// Mitsubishi GX Works2 project: LG 250T Press 3 21.07.21   PLC: Q03UD
// LG 250T Press 3 21.07.21

PROGRAM MAIN
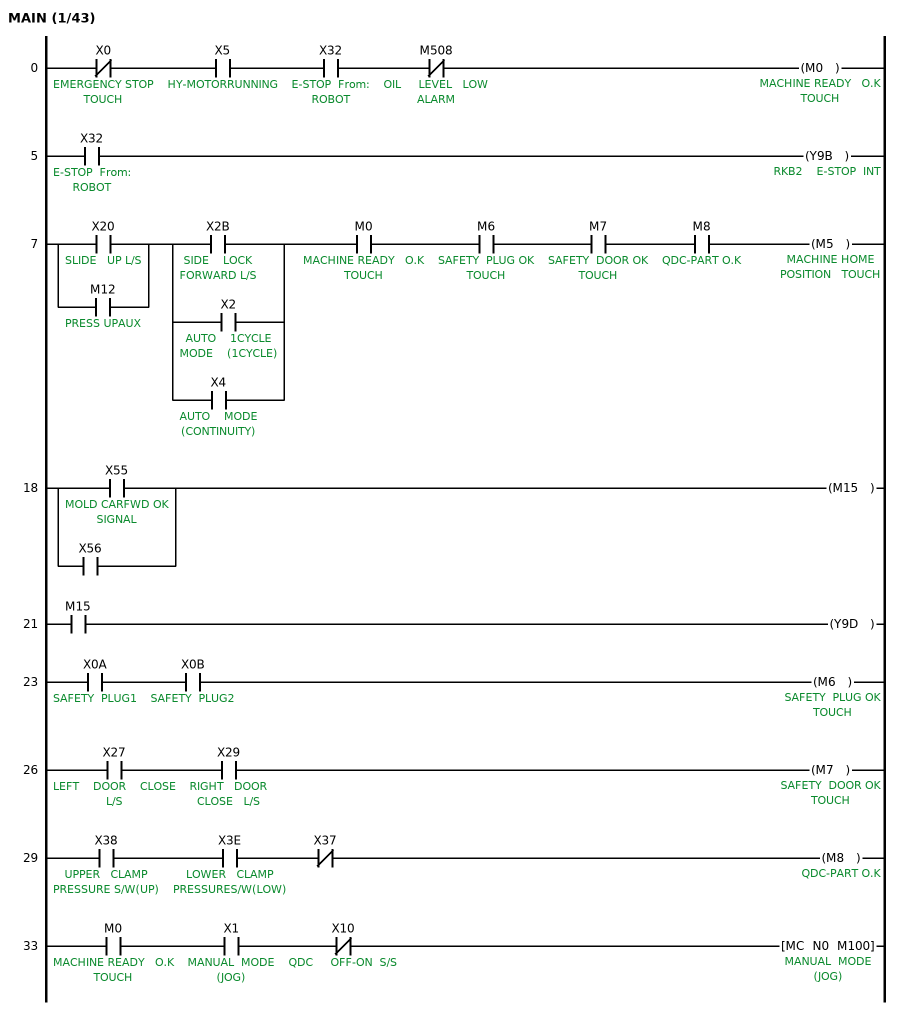
0     LDI     X0  ; EMERGENCY STOP  TOUCH
      AND     X5  ; HY-MOTORRUNNING
      AND     X32  ; E-STOP  From:   ROBOT
      ANI     M508  ; OIL     LEVEL   LOW     ALARM
      OUT     M0  ; MACHINE READY   O.K     TOUCH
5     LD      X32  ; E-STOP  From:   ROBOT
      OUT     Y9B  ; RKB2    E-STOP  INT
7     LD      X20  ; SLIDE   UP L/S
      OR      M12  ; PRESS UPAUX
      LD      X2B  ; SIDE    LOCK    FORWARD L/S
      OR      X2  ; AUTO    1CYCLE  MODE    (1CYCLE)
      OR      X4  ; AUTO    MODE    (CONTINUITY)
      ANB
      AND     M0  ; MACHINE READY   O.K     TOUCH
      AND     M6  ; SAFETY  PLUG OK TOUCH
      AND     M7  ; SAFETY  DOOR OK TOUCH
      AND     M8  ; QDC-PART O.K
      OUT     M5  ; MACHINE HOME POSITION   TOUCH
18    LD      X55  ; MOLD CARFWD OK  SIGNAL
      OR      X56
      OUT     M15
21    LD      M15
      OUT     Y9D
23    LD      X0A  ; SAFETY  PLUG1
      AND     X0B  ; SAFETY  PLUG2
      OUT     M6  ; SAFETY  PLUG OK TOUCH
26    LD      X27  ; LEFT    DOOR    CLOSE   L/S
      AND     X29  ; RIGHT   DOOR    CLOSE   L/S
      OUT     M7  ; SAFETY  DOOR OK TOUCH
29    LD      X38  ; UPPER   CLAMP   PRESSURE S/W(UP)
      AND     X3E  ; LOWER   CLAMP   PRESSURES/W(LOW)
      ANI     X37
      OUT     M8  ; QDC-PART O.K
33    LD      M0  ; MACHINE READY   O.K     TOUCH
      AND     X1  ; MANUAL  MODE    (JOG)
      ANI     X10  ; QDC     OFF-ON  S/S
      MC      N0 M100  ; MANUAL  MODE    (JOG)
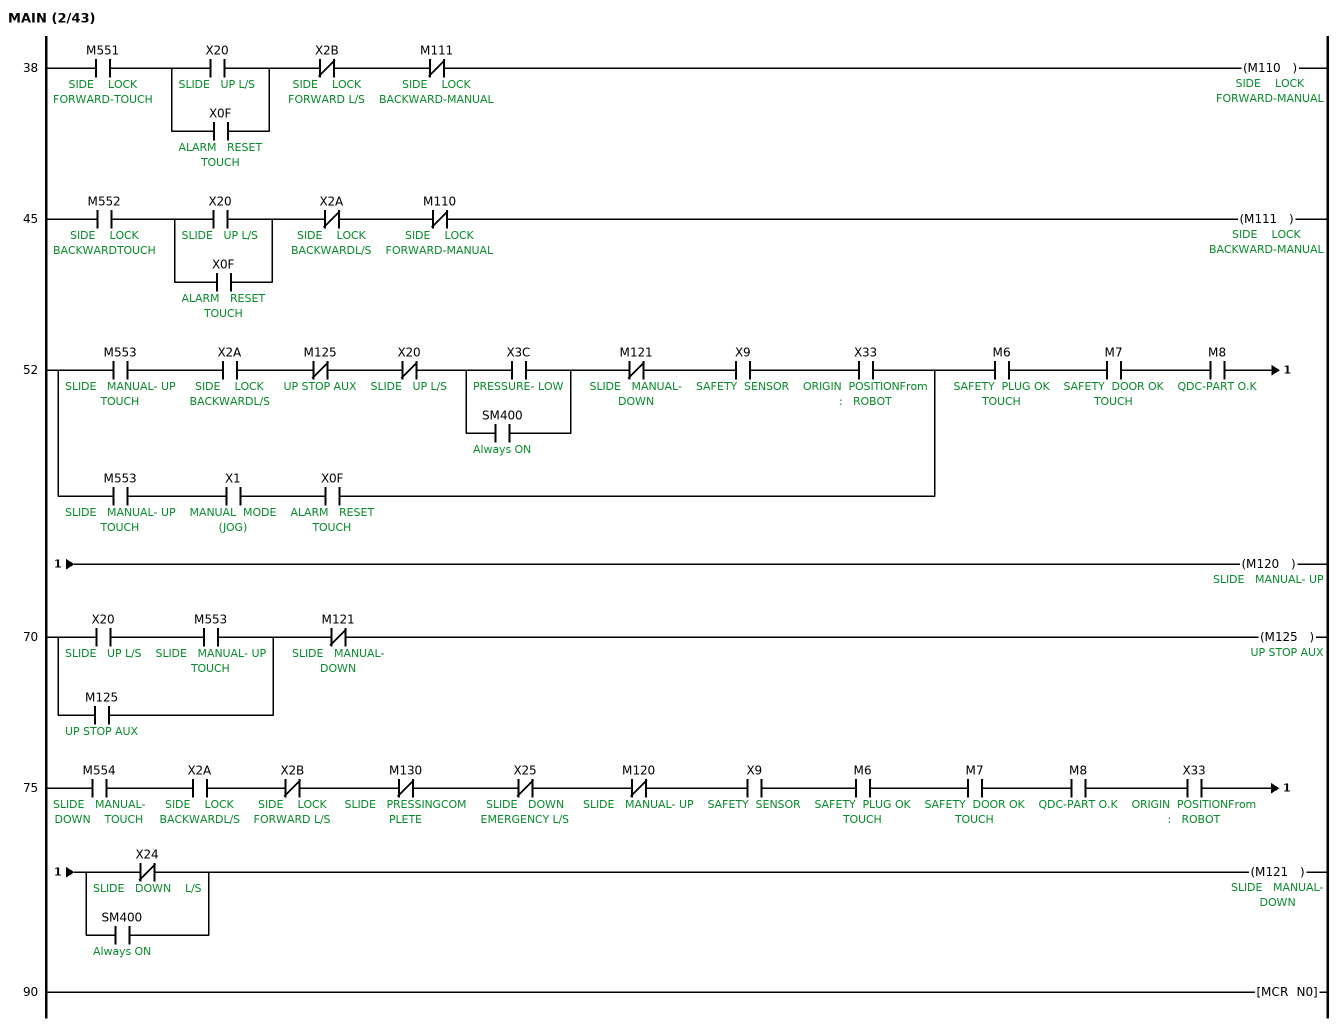
38    LD      M551  ; SIDE    LOCK    FORWARD-TOUCH
      LD      X20  ; SLIDE   UP L/S
      OR      X0F  ; ALARM   RESET   TOUCH
      ANB
      ANI     X2B  ; SIDE    LOCK    FORWARD L/S
      ANI     M111  ; SIDE    LOCK    BACKWARD-MANUAL
      OUT     M110  ; SIDE    LOCK    FORWARD-MANUAL
45    LD      M552  ; SIDE    LOCK    BACKWARDTOUCH
      LD      X20  ; SLIDE   UP L/S
      OR      X0F  ; ALARM   RESET   TOUCH
      ANB
      ANI     X2A  ; SIDE    LOCK    BACKWARDL/S
      ANI     M110  ; SIDE    LOCK    FORWARD-MANUAL
      OUT     M111  ; SIDE    LOCK    BACKWARD-MANUAL
52    LD      M553  ; SLIDE   MANUAL- UP      TOUCH
      AND     X2A  ; SIDE    LOCK    BACKWARDL/S
      ANI     M125  ; UP STOP AUX
      ANI     X20  ; SLIDE   UP L/S
      LD      X3C  ; PRESSURE- LOW
      OR      SM400  ; Always ON
      ANB
      ANI     M121  ; SLIDE   MANUAL- DOWN
      AND     X9  ; SAFETY  SENSOR
      AND     X33  ; ORIGIN  POSITIONFrom:   ROBOT
      LD      M553  ; SLIDE   MANUAL- UP      TOUCH
      AND     X1  ; MANUAL  MODE    (JOG)
      AND     X0F  ; ALARM   RESET   TOUCH
      ORB
      AND     M6  ; SAFETY  PLUG OK TOUCH
      AND     M7  ; SAFETY  DOOR OK TOUCH
      AND     M8  ; QDC-PART O.K
      OUT     M120  ; SLIDE   MANUAL- UP
70    LD      X20  ; SLIDE   UP L/S
      AND     M553  ; SLIDE   MANUAL- UP      TOUCH
      OR      M125  ; UP STOP AUX
      ANI     M121  ; SLIDE   MANUAL- DOWN
      OUT     M125  ; UP STOP AUX
75    LD      M554  ; SLIDE   MANUAL- DOWN    TOUCH
      AND     X2A  ; SIDE    LOCK    BACKWARDL/S
      ANI     X2B  ; SIDE    LOCK    FORWARD L/S
      ANI     M130  ; SLIDE   PRESSINGCOMPLETE
      ANI     X25  ; SLIDE   DOWN    EMERGENCY L/S
      ANI     M120  ; SLIDE   MANUAL- UP
      AND     X9  ; SAFETY  SENSOR
      AND     M6  ; SAFETY  PLUG OK TOUCH
      AND     M7  ; SAFETY  DOOR OK TOUCH
      AND     M8  ; QDC-PART O.K
      AND     X33  ; ORIGIN  POSITIONFrom:   ROBOT
      LDI     X24  ; SLIDE   DOWN    L/S
      OR      SM400  ; Always ON
      ANB
      OUT     M121  ; SLIDE   MANUAL- DOWN
90    MCR     N0
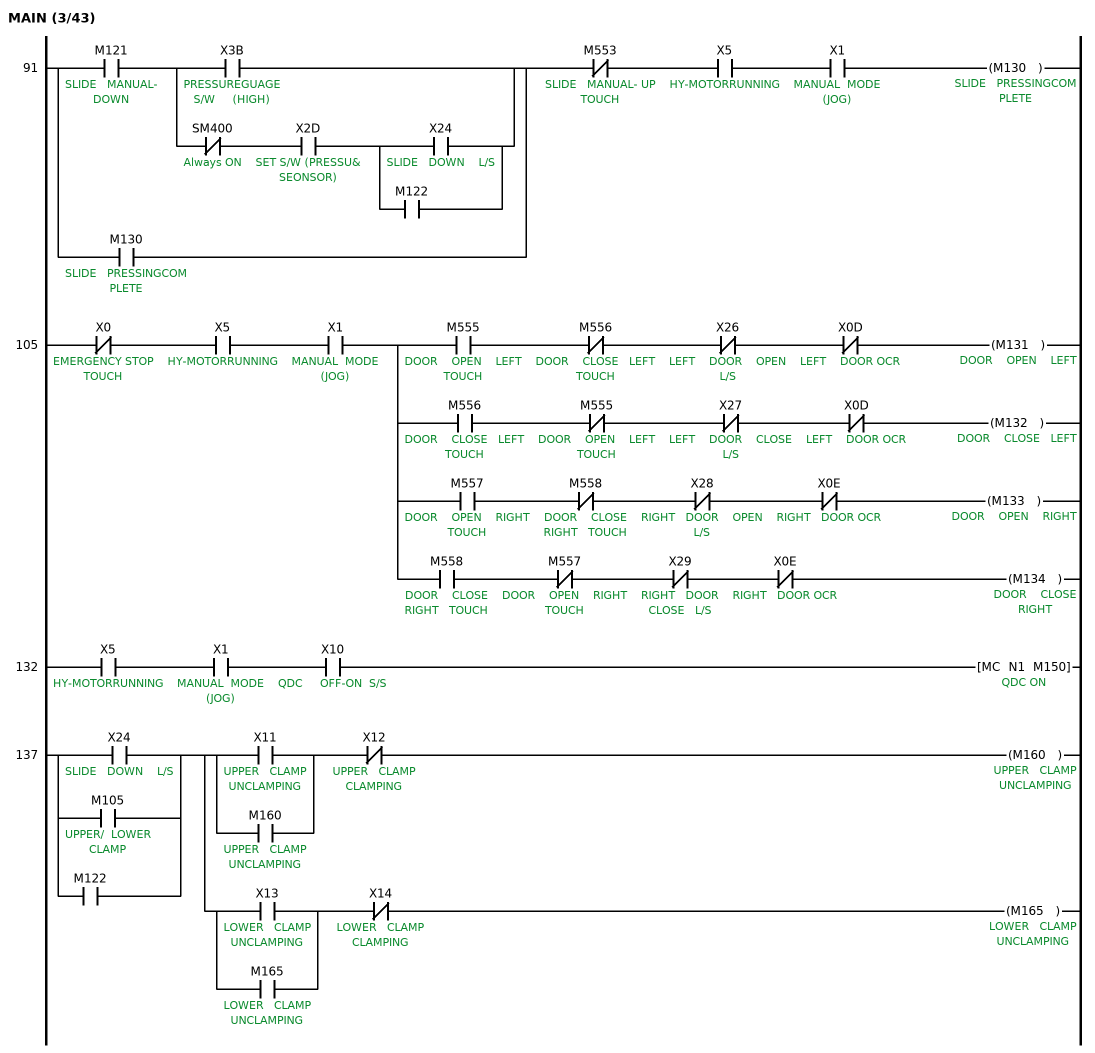
91    LD      M121  ; SLIDE   MANUAL- DOWN
      LD      X3B  ; PRESSUREGUAGE   S/W     (HIGH)
      LDI     SM400  ; Always ON
      AND     X2D  ; SET S/W (PRESSU& SEONSOR)
      LD      X24  ; SLIDE   DOWN    L/S
      OR      M122
      ANB
      ORB
      ANB
      OR      M130  ; SLIDE   PRESSINGCOMPLETE
      ANI     M553  ; SLIDE   MANUAL- UP      TOUCH
      AND     X5  ; HY-MOTORRUNNING
      AND     X1  ; MANUAL  MODE    (JOG)
      OUT     M130  ; SLIDE   PRESSINGCOMPLETE
105   LDI     X0  ; EMERGENCY STOP  TOUCH
      AND     X5  ; HY-MOTORRUNNING
      AND     X1  ; MANUAL  MODE    (JOG)
      MPS
      AND     M555  ; DOOR    OPEN    LEFT    TOUCH
      ANI     M556  ; DOOR    CLOSE   LEFT    TOUCH
      ANI     X26  ; LEFT    DOOR    OPEN L/S
      ANI     X0D  ; LEFT    DOOR OCR
      OUT     M131  ; DOOR    OPEN    LEFT
      MRD
      AND     M556  ; DOOR    CLOSE   LEFT    TOUCH
      ANI     M555  ; DOOR    OPEN    LEFT    TOUCH
      ANI     X27  ; LEFT    DOOR    CLOSE   L/S
      ANI     X0D  ; LEFT    DOOR OCR
      OUT     M132  ; DOOR    CLOSE   LEFT
      MRD
      AND     M557  ; DOOR    OPEN    RIGHT   TOUCH
      ANI     M558  ; DOOR    CLOSE   RIGHT   TOUCH
      ANI     X28  ; RIGHT   DOOR    OPEN L/S
      ANI     X0E  ; RIGHT   DOOR OCR
      OUT     M133  ; DOOR    OPEN    RIGHT
      MPP
      AND     M558  ; DOOR    CLOSE   RIGHT   TOUCH
      ANI     M557  ; DOOR    OPEN    RIGHT   TOUCH
      ANI     X29  ; RIGHT   DOOR    CLOSE   L/S
      ANI     X0E  ; RIGHT   DOOR OCR
      OUT     M134  ; DOOR    CLOSE   RIGHT
132   LD      X5  ; HY-MOTORRUNNING
      AND     X1  ; MANUAL  MODE    (JOG)
      AND     X10  ; QDC     OFF-ON  S/S
      MC      N1 M150  ; QDC ON
137   LD      X24  ; SLIDE   DOWN    L/S
      OR      M105  ; UPPER/  LOWER   CLAMP
      OR      M122
      MPS
      LD      X11  ; UPPER   CLAMP   UNCLAMPING
      OR      M160  ; UPPER   CLAMP   UNCLAMPING
      ANB
      ANI     X12  ; UPPER   CLAMP   CLAMPING
      OUT     M160  ; UPPER   CLAMP   UNCLAMPING
      MPP
      LD      X13  ; LOWER   CLAMP   UNCLAMPING
      OR      M165  ; LOWER   CLAMP   UNCLAMPING
      ANB
      ANI     X14  ; LOWER   CLAMP   CLAMPING
      OUT     M165  ; LOWER   CLAMP   UNCLAMPING
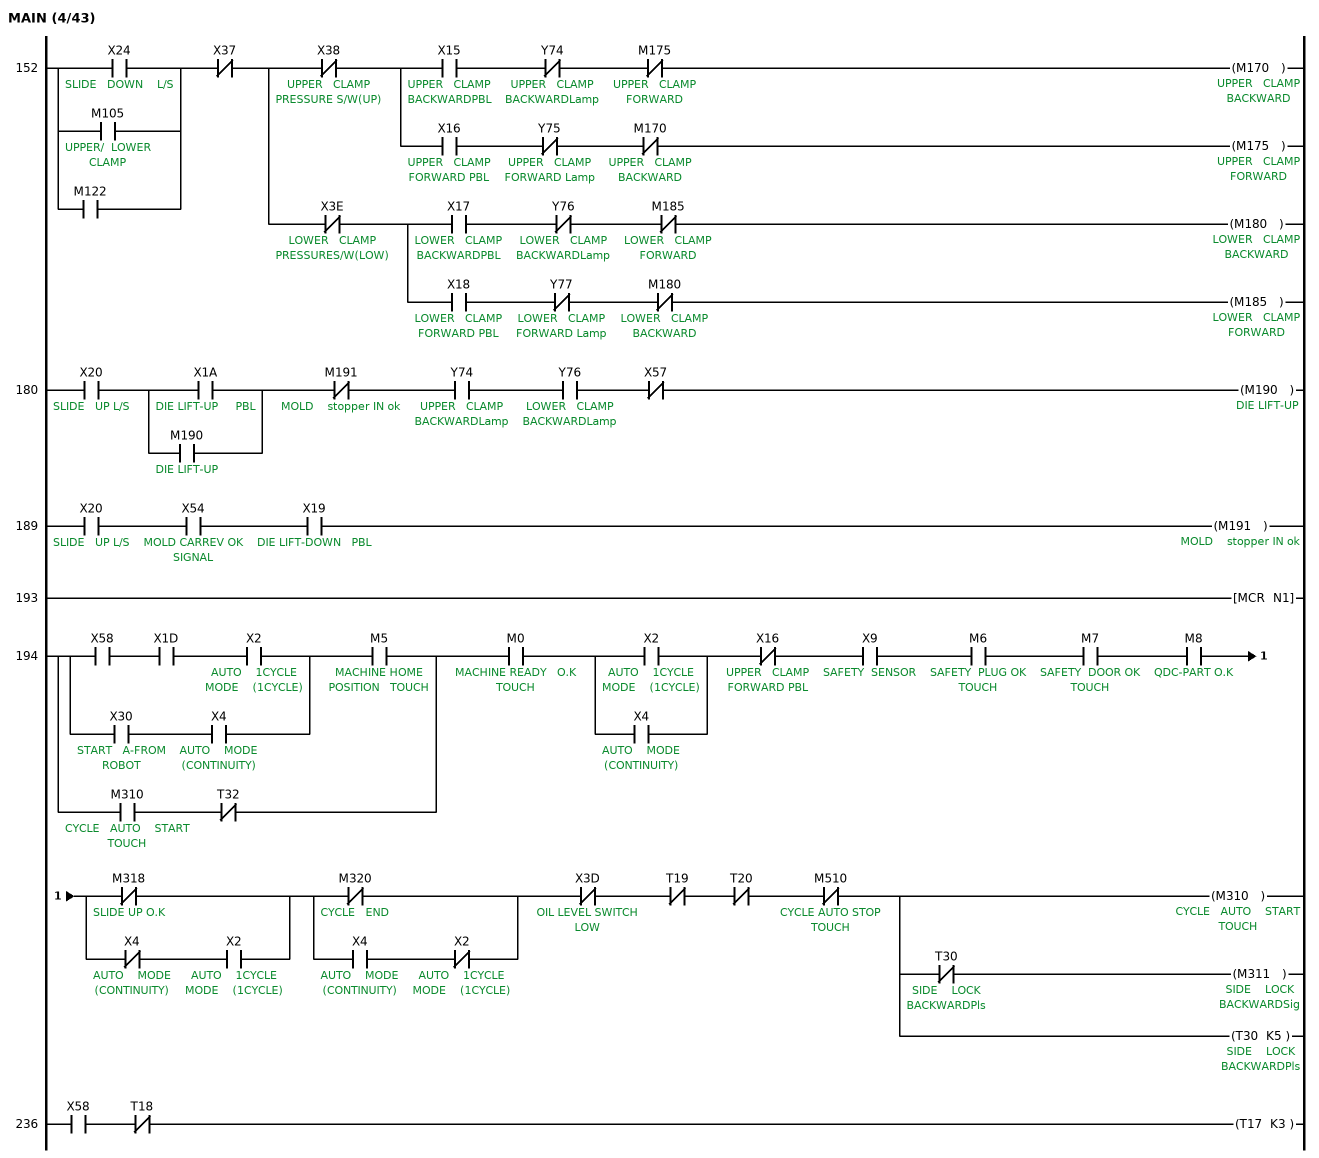
152   LD      X24  ; SLIDE   DOWN    L/S
      OR      M105  ; UPPER/  LOWER   CLAMP
      OR      M122
      ANI     X37
      MPS
      ANI     X38  ; UPPER   CLAMP   PRESSURE S/W(UP)
      MPS
      AND     X15  ; UPPER   CLAMP   BACKWARDPBL
      ANI     Y74  ; UPPER   CLAMP   BACKWARDLamp
      ANI     M175  ; UPPER   CLAMP   FORWARD
      OUT     M170  ; UPPER   CLAMP   BACKWARD
      MPP
      AND     X16  ; UPPER   CLAMP   FORWARD PBL
      ANI     Y75  ; UPPER   CLAMP   FORWARD Lamp
      ANI     M170  ; UPPER   CLAMP   BACKWARD
      OUT     M175  ; UPPER   CLAMP   FORWARD
      MPP
      ANI     X3E  ; LOWER   CLAMP   PRESSURES/W(LOW)
      MPS
      AND     X17  ; LOWER   CLAMP   BACKWARDPBL
      ANI     Y76  ; LOWER   CLAMP   BACKWARDLamp
      ANI     M185  ; LOWER   CLAMP   FORWARD
      OUT     M180  ; LOWER   CLAMP   BACKWARD
      MPP
      AND     X18  ; LOWER   CLAMP   FORWARD PBL
      ANI     Y77  ; LOWER   CLAMP   FORWARD Lamp
      ANI     M180  ; LOWER   CLAMP   BACKWARD
      OUT     M185  ; LOWER   CLAMP   FORWARD
180   LD      X20  ; SLIDE   UP L/S
      LD      X1A  ; DIE LIFT-UP     PBL
      OR      M190  ; DIE LIFT-UP
      ANB
      ANI     M191  ; MOLD    stopper IN ok
      AND     Y74  ; UPPER   CLAMP   BACKWARDLamp
      AND     Y76  ; LOWER   CLAMP   BACKWARDLamp
      ANI     X57
      OUT     M190  ; DIE LIFT-UP
189   LD      X20  ; SLIDE   UP L/S
      AND     X54  ; MOLD CARREV OK  SIGNAL
      AND     X19  ; DIE LIFT-DOWN   PBL
      OUT     M191  ; MOLD    stopper IN ok
193   MCR     N1
194   LD      X58
      AND     X1D
      AND     X2  ; AUTO    1CYCLE  MODE    (1CYCLE)
      LD      X30  ; START   A-FROM  ROBOT
      AND     X4  ; AUTO    MODE    (CONTINUITY)
      ORB
      AND     M5  ; MACHINE HOME POSITION   TOUCH
      LD      M310  ; CYCLE   AUTO    START   TOUCH
      ANI     T32
      ORB
      AND     M0  ; MACHINE READY   O.K     TOUCH
      LD      X2  ; AUTO    1CYCLE  MODE    (1CYCLE)
      OR      X4  ; AUTO    MODE    (CONTINUITY)
      ANB
      ANI     X16  ; UPPER   CLAMP   FORWARD PBL
      AND     X9  ; SAFETY  SENSOR
      AND     M6  ; SAFETY  PLUG OK TOUCH
      AND     M7  ; SAFETY  DOOR OK TOUCH
      AND     M8  ; QDC-PART O.K
      LDI     M318  ; SLIDE UP O.K
      LDI     X4  ; AUTO    MODE    (CONTINUITY)
      AND     X2  ; AUTO    1CYCLE  MODE    (1CYCLE)
      ORB
      ANB
      LDI     M320  ; CYCLE   END
      LD      X4  ; AUTO    MODE    (CONTINUITY)
      ANI     X2  ; AUTO    1CYCLE  MODE    (1CYCLE)
      ORB
      ANB
      ANI     X3D  ; OIL LEVEL SWITCH LOW
      ANI     T19
      ANI     T20
      ANI     M510  ; CYCLE AUTO STOP TOUCH
      OUT     M310  ; CYCLE   AUTO    START   TOUCH
      MPS
      ANI     T30  ; SIDE    LOCK    BACKWARDPls
      OUT     M311  ; SIDE    LOCK    BACKWARDSig
      MPP
      OUT     T30 K5  ; SIDE    LOCK    BACKWARDPls
236   LD      X58
      ANI     T18
      OUT     T17 K3
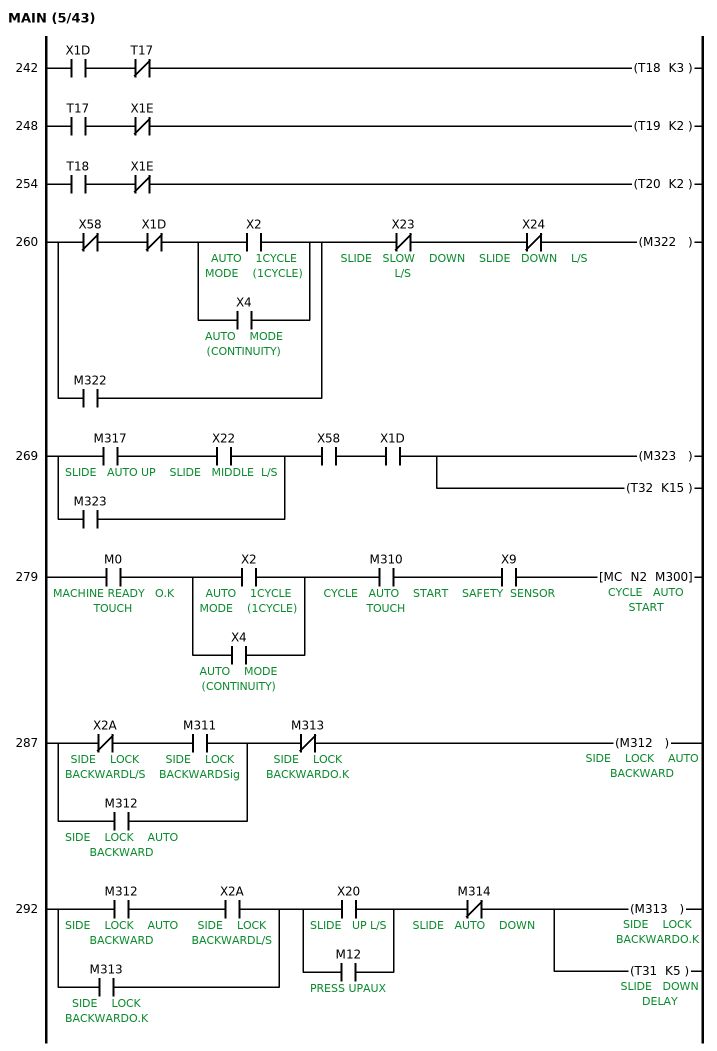
242   LD      X1D
      ANI     T17
      OUT     T18 K3
248   LD      T17
      ANI     X1E
      OUT     T19 K2
254   LD      T18
      ANI     X1E
      OUT     T20 K2
260   LDI     X58
      ANI     X1D
      LD      X2  ; AUTO    1CYCLE  MODE    (1CYCLE)
      OR      X4  ; AUTO    MODE    (CONTINUITY)
      ANB
      OR      M322
      ANI     X23  ; SLIDE   SLOW    DOWN L/S
      ANI     X24  ; SLIDE   DOWN    L/S
      OUT     M322
269   LD      M317  ; SLIDE   AUTO UP
      AND     X22  ; SLIDE   MIDDLE  L/S
      OR      M323
      AND     X58
      AND     X1D
      OUT     M323
      OUT     T32 K15
279   LD      M0  ; MACHINE READY   O.K     TOUCH
      LD      X2  ; AUTO    1CYCLE  MODE    (1CYCLE)
      OR      X4  ; AUTO    MODE    (CONTINUITY)
      ANB
      AND     M310  ; CYCLE   AUTO    START   TOUCH
      AND     X9  ; SAFETY  SENSOR
      MC      N2 M300  ; CYCLE   AUTO    START
287   LDI     X2A  ; SIDE    LOCK    BACKWARDL/S
      AND     M311  ; SIDE    LOCK    BACKWARDSig
      OR      M312  ; SIDE    LOCK    AUTO    BACKWARD
      ANI     M313  ; SIDE    LOCK    BACKWARDO.K
      OUT     M312  ; SIDE    LOCK    AUTO    BACKWARD
292   LD      M312  ; SIDE    LOCK    AUTO    BACKWARD
      AND     X2A  ; SIDE    LOCK    BACKWARDL/S
      OR      M313  ; SIDE    LOCK    BACKWARDO.K
      LD      X20  ; SLIDE   UP L/S
      OR      M12  ; PRESS UPAUX
      ANB
      ANI     M314  ; SLIDE   AUTO    DOWN
      OUT     M313  ; SIDE    LOCK    BACKWARDO.K
      OUT     T31 K5  ; SLIDE   DOWN    DELAY
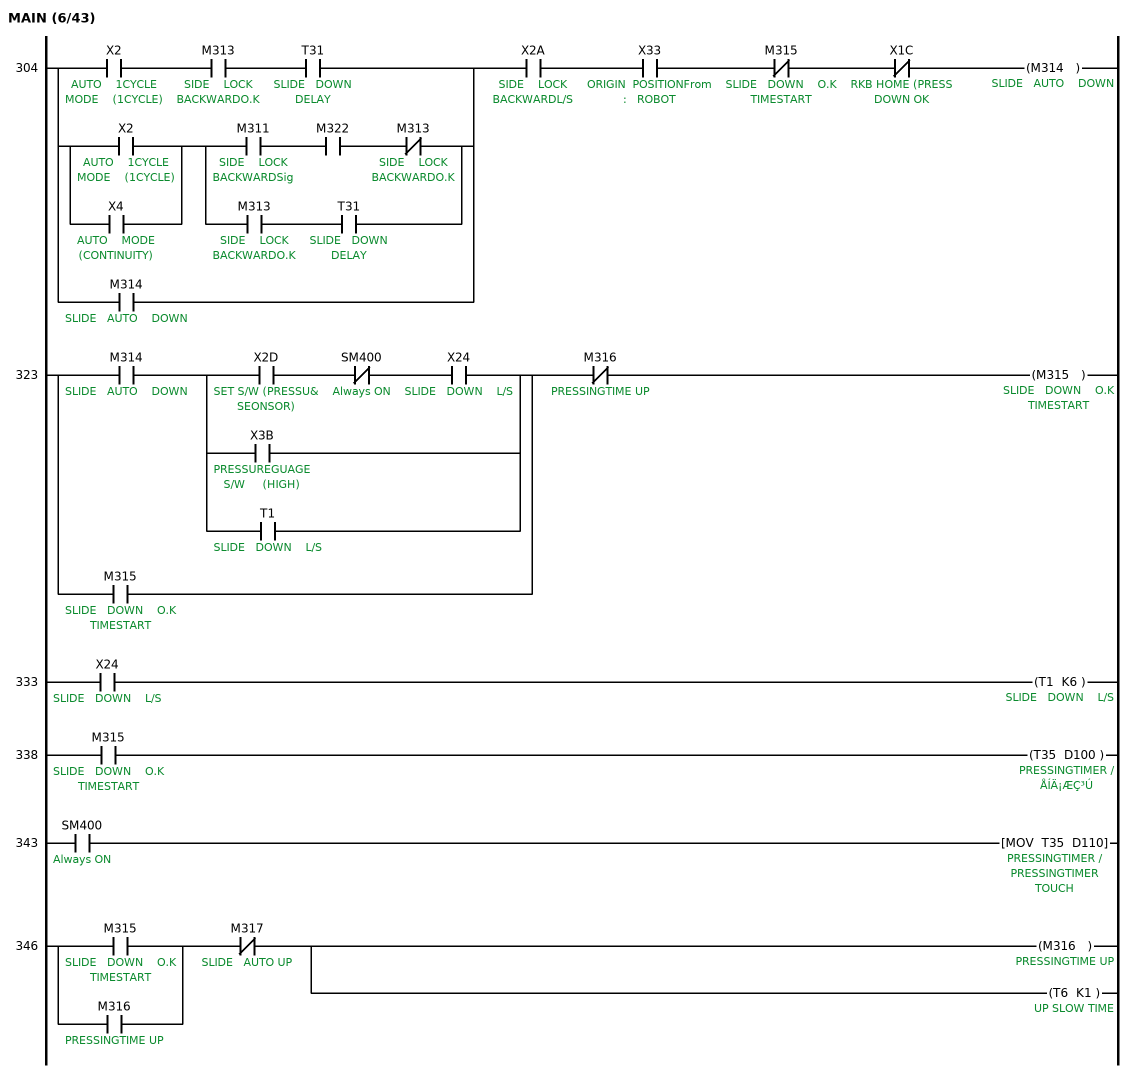
304   LD      X2  ; AUTO    1CYCLE  MODE    (1CYCLE)
      AND     M313  ; SIDE    LOCK    BACKWARDO.K
      AND     T31  ; SLIDE   DOWN    DELAY
      LD      X2  ; AUTO    1CYCLE  MODE    (1CYCLE)
      OR      X4  ; AUTO    MODE    (CONTINUITY)
      LD      M311  ; SIDE    LOCK    BACKWARDSig
      AND     M322
      ANI     M313  ; SIDE    LOCK    BACKWARDO.K
      LD      M313  ; SIDE    LOCK    BACKWARDO.K
      AND     T31  ; SLIDE   DOWN    DELAY
      ORB
      ANB
      ORB
      OR      M314  ; SLIDE   AUTO    DOWN
      AND     X2A  ; SIDE    LOCK    BACKWARDL/S
      AND     X33  ; ORIGIN  POSITIONFrom:   ROBOT
      ANI     M315  ; SLIDE   DOWN    O.K TIMESTART
      ANI     X1C  ; RKB HOME (PRESS DOWN OK
      OUT     M314  ; SLIDE   AUTO    DOWN
323   LD      M314  ; SLIDE   AUTO    DOWN
      LD      X2D  ; SET S/W (PRESSU& SEONSOR)
      ANI     SM400  ; Always ON
      AND     X24  ; SLIDE   DOWN    L/S
      OR      X3B  ; PRESSUREGUAGE   S/W     (HIGH)
      OR      T1  ; SLIDE   DOWN    L/S
      ANB
      OR      M315  ; SLIDE   DOWN    O.K TIMESTART
      ANI     M316  ; PRESSINGTIME UP
      OUT     M315  ; SLIDE   DOWN    O.K TIMESTART
333   LD      X24  ; SLIDE   DOWN    L/S
      OUT     T1 K6  ; SLIDE   DOWN    L/S
338   LD      M315  ; SLIDE   DOWN    O.K TIMESTART
      OUT     T35 D100  ; PRESSINGTIMER / ÅÍÄ¡ÆÇ³Ú
343   LD      SM400  ; Always ON
      MOV     T35 D110  ; PRESSINGTIMER   TOUCH
346   LD      M315  ; SLIDE   DOWN    O.K TIMESTART
      OR      M316  ; PRESSINGTIME UP
      ANI     M317  ; SLIDE   AUTO UP
      OUT     M316  ; PRESSINGTIME UP
      OUT     T6 K1  ; UP SLOW TIME
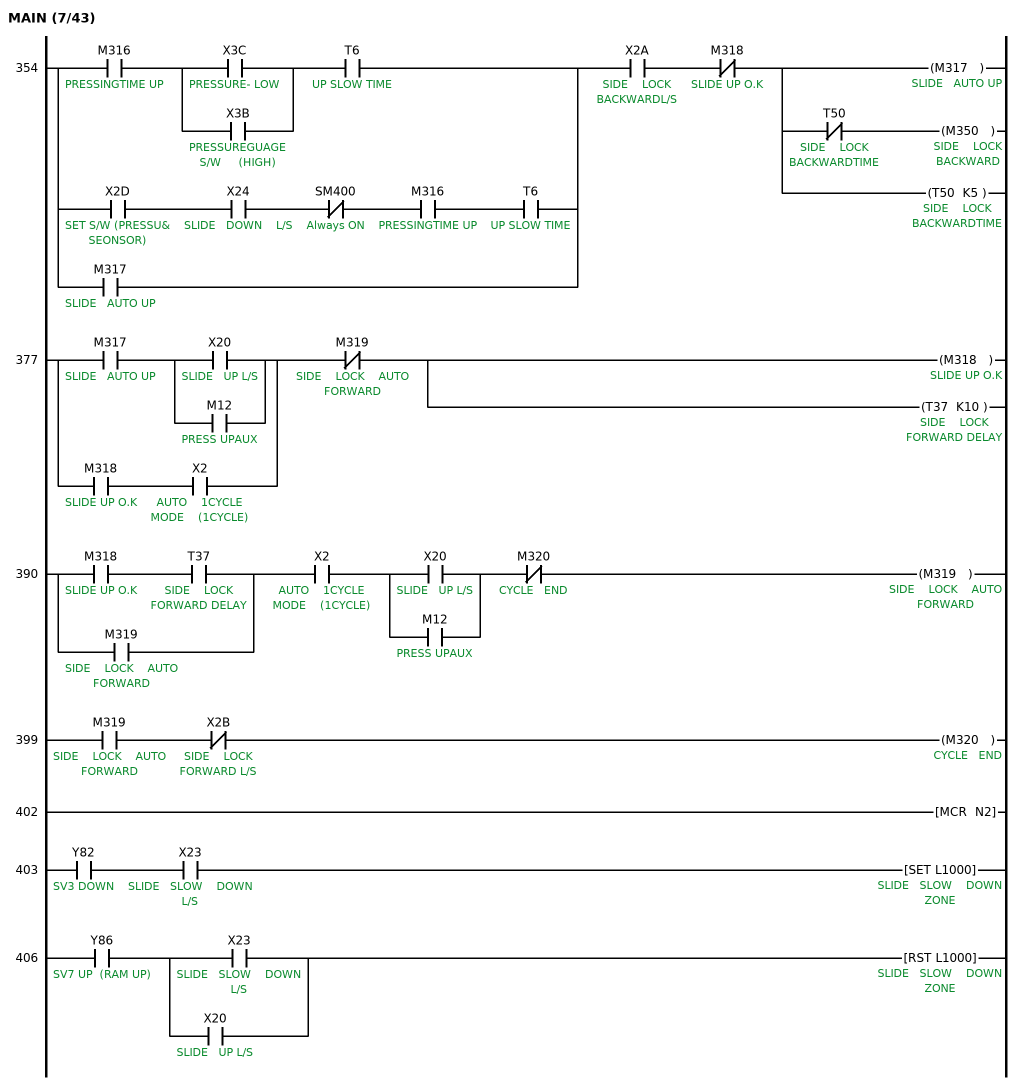
354   LD      M316  ; PRESSINGTIME UP
      LD      X3C  ; PRESSURE- LOW
      OR      X3B  ; PRESSUREGUAGE   S/W     (HIGH)
      ANB
      AND     T6  ; UP SLOW TIME
      LD      X2D  ; SET S/W (PRESSU& SEONSOR)
      AND     X24  ; SLIDE   DOWN    L/S
      ANI     SM400  ; Always ON
      AND     M316  ; PRESSINGTIME UP
      AND     T6  ; UP SLOW TIME
      ORB
      OR      M317  ; SLIDE   AUTO UP
      AND     X2A  ; SIDE    LOCK    BACKWARDL/S
      ANI     M318  ; SLIDE UP O.K
      OUT     M317  ; SLIDE   AUTO UP
      MPS
      ANI     T50  ; SIDE    LOCK    BACKWARDTIME
      OUT     M350  ; SIDE    LOCK    BACKWARD
      MPP
      OUT     T50 K5  ; SIDE    LOCK    BACKWARDTIME
377   LD      M317  ; SLIDE   AUTO UP
      LD      X20  ; SLIDE   UP L/S
      OR      M12  ; PRESS UPAUX
      ANB
      LD      M318  ; SLIDE UP O.K
      AND     X2  ; AUTO    1CYCLE  MODE    (1CYCLE)
      ORB
      ANI     M319  ; SIDE    LOCK    AUTO    FORWARD
      OUT     M318  ; SLIDE UP O.K
      OUT     T37 K10  ; SIDE    LOCK    FORWARD DELAY
390   LD      M318  ; SLIDE UP O.K
      AND     T37  ; SIDE    LOCK    FORWARD DELAY
      OR      M319  ; SIDE    LOCK    AUTO    FORWARD
      AND     X2  ; AUTO    1CYCLE  MODE    (1CYCLE)
      LD      X20  ; SLIDE   UP L/S
      OR      M12  ; PRESS UPAUX
      ANB
      ANI     M320  ; CYCLE   END
      OUT     M319  ; SIDE    LOCK    AUTO    FORWARD
399   LD      M319  ; SIDE    LOCK    AUTO    FORWARD
      ANI     X2B  ; SIDE    LOCK    FORWARD L/S
      OUT     M320  ; CYCLE   END
402   MCR     N2
403   LD      Y82  ; SV3 DOWN
      AND     X23  ; SLIDE   SLOW    DOWN L/S
      SET     L1000  ; SLIDE   SLOW    DOWN    ZONE
406   LD      Y86  ; SV7 UP  (RAM UP)
      LD      X23  ; SLIDE   SLOW    DOWN L/S
      OR      X20  ; SLIDE   UP L/S
      ANB
      RST     L1000  ; SLIDE   SLOW    DOWN    ZONE
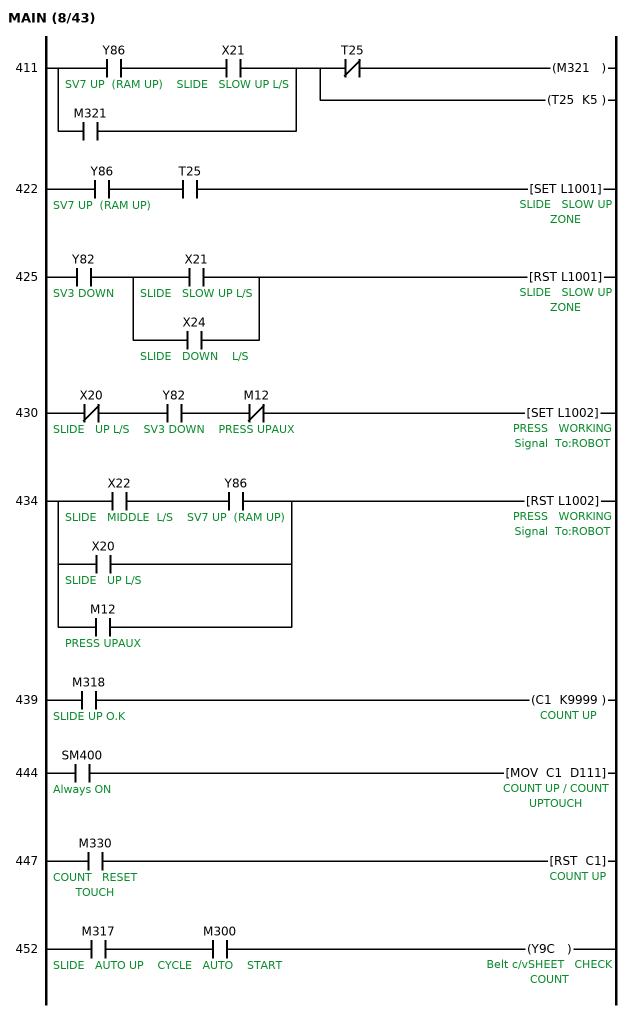
411   LD      Y86  ; SV7 UP  (RAM UP)
      AND     X21  ; SLIDE   SLOW UP L/S
      OR      M321
      MPS
      ANI     T25
      OUT     M321
      MPP
      OUT     T25 K5
422   LD      Y86  ; SV7 UP  (RAM UP)
      AND     T25
      SET     L1001  ; SLIDE   SLOW UP ZONE
425   LD      Y82  ; SV3 DOWN
      LD      X21  ; SLIDE   SLOW UP L/S
      OR      X24  ; SLIDE   DOWN    L/S
      ANB
      RST     L1001  ; SLIDE   SLOW UP ZONE
430   LDI     X20  ; SLIDE   UP L/S
      AND     Y82  ; SV3 DOWN
      ANI     M12  ; PRESS UPAUX
      SET     L1002  ; PRESS   WORKING Signal  To:ROBOT
434   LD      X22  ; SLIDE   MIDDLE  L/S
      AND     Y86  ; SV7 UP  (RAM UP)
      OR      X20  ; SLIDE   UP L/S
      OR      M12  ; PRESS UPAUX
      RST     L1002  ; PRESS   WORKING Signal  To:ROBOT
439   LD      M318  ; SLIDE UP O.K
      OUT     C1 K9999  ; COUNT UP
444   LD      SM400  ; Always ON
      MOV     C1 D111  ; COUNT UPTOUCH
447   LD      M330  ; COUNT   RESET   TOUCH
      RST     C1  ; COUNT UP
452   LD      M317  ; SLIDE   AUTO UP
      AND     M300  ; CYCLE   AUTO    START
      OUT     Y9C  ; Belt c/vSHEET   CHECK   COUNT
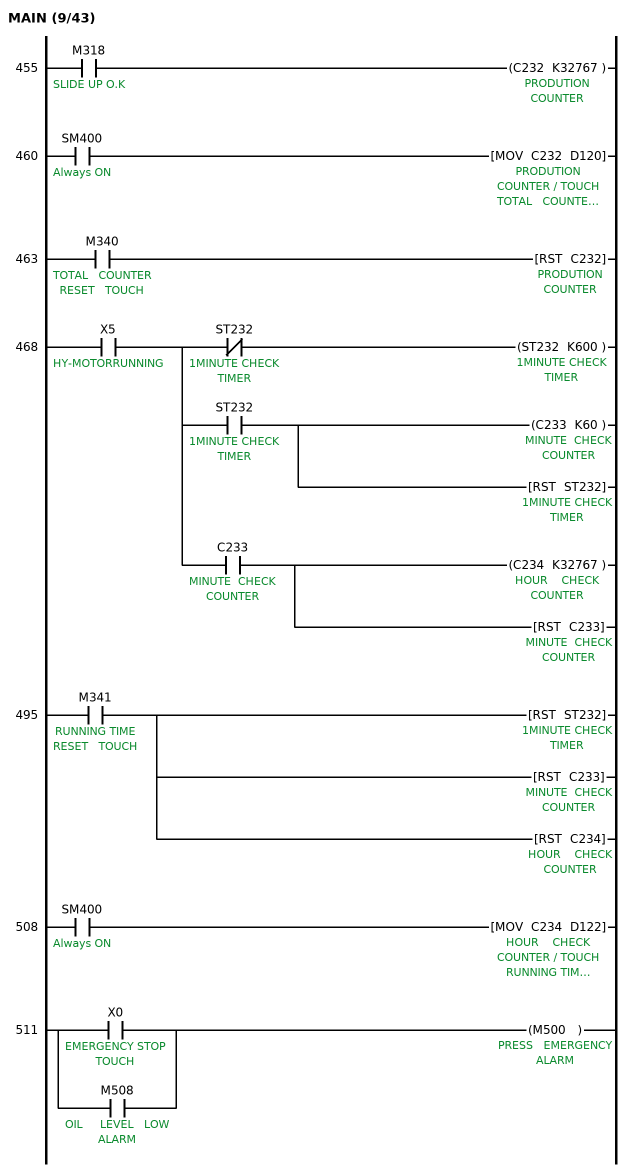
455   LD      M318  ; SLIDE UP O.K
      OUT     C232 K32767  ; PRODUTION       COUNTER
460   LD      SM400  ; Always ON
      MOV     C232 D120  ; TOUCH   TOTAL   COUNTER VALUE
463   LD      M340  ; TOTAL   COUNTER RESET   TOUCH
      RST     C232  ; PRODUTION       COUNTER
468   LD      X5  ; HY-MOTORRUNNING
      MPS
      ANI     ST232  ; 1MINUTE CHECK   TIMER
      OUT     ST232 K600  ; 1MINUTE CHECK   TIMER
      MRD
      AND     ST232  ; 1MINUTE CHECK   TIMER
      OUT     C233 K60  ; MINUTE  CHECK   COUNTER
      RST     ST232  ; 1MINUTE CHECK   TIMER
      MPP
      AND     C233  ; MINUTE  CHECK   COUNTER
      OUT     C234 K32767  ; HOUR    CHECK   COUNTER
      RST     C233  ; MINUTE  CHECK   COUNTER
495   LD      M341  ; RUNNING TIME    RESET   TOUCH
      RST     ST232  ; 1MINUTE CHECK   TIMER
      RST     C233  ; MINUTE  CHECK   COUNTER
      RST     C234  ; HOUR    CHECK   COUNTER
508   LD      SM400  ; Always ON
      MOV     C234 D122  ; TOUCH   RUNNING TIME    VALUE
511   LD      X0  ; EMERGENCY STOP  TOUCH
      OR      M508  ; OIL     LEVEL   LOW     ALARM
      OUT     M500  ; PRESS   EMERGENCY       ALARM
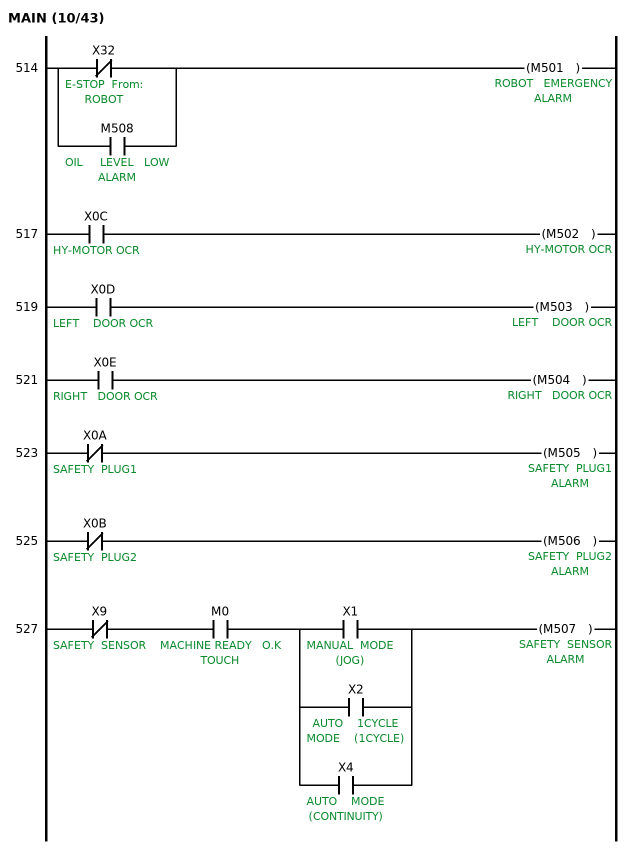
514   LDI     X32  ; E-STOP  From:   ROBOT
      OR      M508  ; OIL     LEVEL   LOW     ALARM
      OUT     M501  ; ROBOT   EMERGENCY       ALARM
517   LD      X0C  ; HY-MOTOR OCR
      OUT     M502  ; HY-MOTOR OCR
519   LD      X0D  ; LEFT    DOOR OCR
      OUT     M503  ; LEFT    DOOR OCR
521   LD      X0E  ; RIGHT   DOOR OCR
      OUT     M504  ; RIGHT   DOOR OCR
523   LDI     X0A  ; SAFETY  PLUG1
      OUT     M505  ; SAFETY  PLUG1   ALARM
525   LDI     X0B  ; SAFETY  PLUG2
      OUT     M506  ; SAFETY  PLUG2   ALARM
527   LDI     X9  ; SAFETY  SENSOR
      AND     M0  ; MACHINE READY   O.K     TOUCH
      LD      X1  ; MANUAL  MODE    (JOG)
      OR      X2  ; AUTO    1CYCLE  MODE    (1CYCLE)
      OR      X4  ; AUTO    MODE    (CONTINUITY)
      ANB
      OUT     M507  ; SAFETY  SENSOR  ALARM
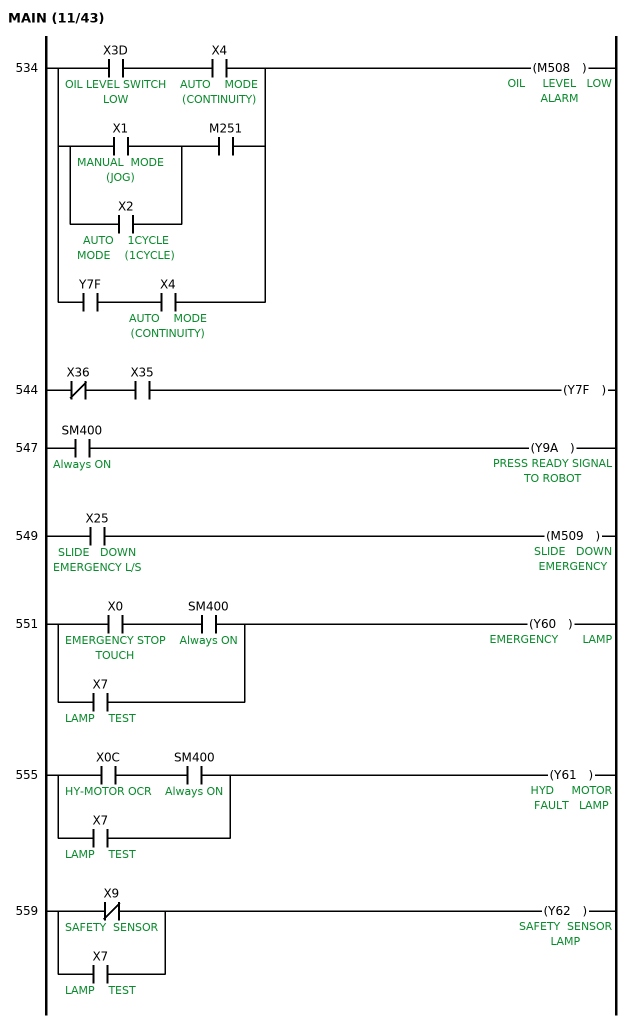
534   LD      X3D  ; OIL LEVEL SWITCH LOW
      AND     X4  ; AUTO    MODE    (CONTINUITY)
      LD      X1  ; MANUAL  MODE    (JOG)
      OR      X2  ; AUTO    1CYCLE  MODE    (1CYCLE)
      AND     M251
      ORB
      LD      Y7F
      AND     X4  ; AUTO    MODE    (CONTINUITY)
      ORB
      OUT     M508  ; OIL     LEVEL   LOW     ALARM
544   LDI     X36
      AND     X35
      OUT     Y7F
547   LD      SM400  ; Always ON
      OUT     Y9A  ; PRESS READY SIGNAL TO ROBOT
549   LD      X25  ; SLIDE   DOWN    EMERGENCY L/S
      OUT     M509  ; SLIDE   DOWN    EMERGENCY
551   LD      X0  ; EMERGENCY STOP  TOUCH
      AND     SM400  ; Always ON
      OR      X7  ; LAMP    TEST
      OUT     Y60  ; EMERGENCY       LAMP
555   LD      X0C  ; HY-MOTOR OCR
      AND     SM400  ; Always ON
      OR      X7  ; LAMP    TEST
      OUT     Y61  ; HYD     MOTOR   FAULT   LAMP
559   LDI     X9  ; SAFETY  SENSOR
      OR      X7  ; LAMP    TEST
      OUT     Y62  ; SAFETY  SENSOR  LAMP
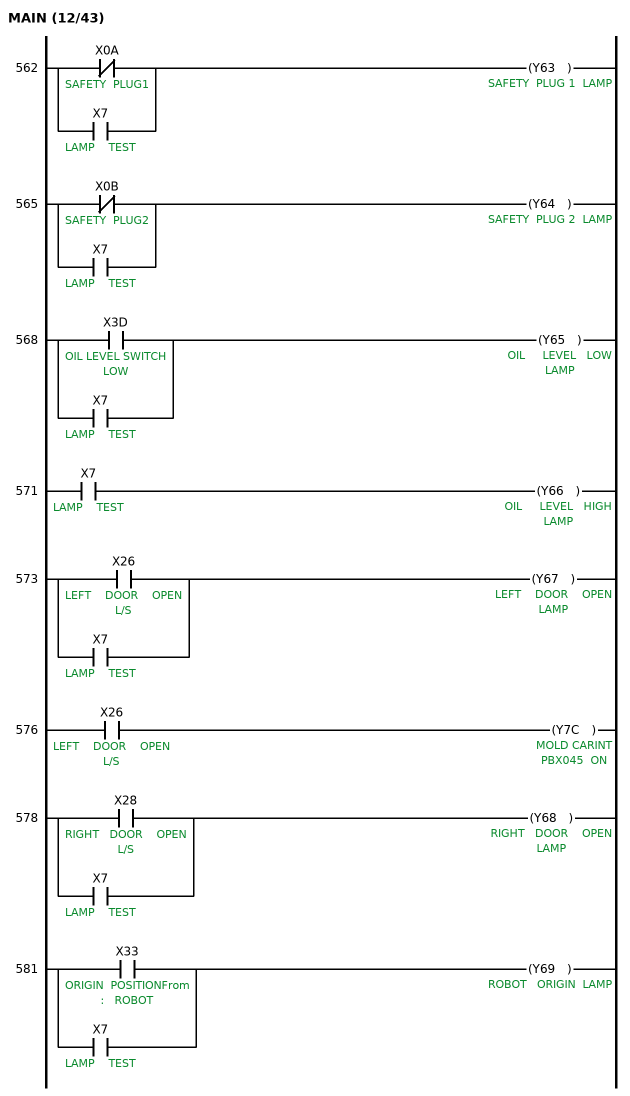
562   LDI     X0A  ; SAFETY  PLUG1
      OR      X7  ; LAMP    TEST
      OUT     Y63  ; SAFETY  PLUG 1  LAMP
565   LDI     X0B  ; SAFETY  PLUG2
      OR      X7  ; LAMP    TEST
      OUT     Y64  ; SAFETY  PLUG 2  LAMP
568   LD      X3D  ; OIL LEVEL SWITCH LOW
      OR      X7  ; LAMP    TEST
      OUT     Y65  ; OIL     LEVEL   LOW LAMP
571   LD      X7  ; LAMP    TEST
      OUT     Y66  ; OIL     LEVEL   HIGH     LAMP
573   LD      X26  ; LEFT    DOOR    OPEN L/S
      OR      X7  ; LAMP    TEST
      OUT     Y67  ; LEFT    DOOR    OPEN    LAMP
576   LD      X26  ; LEFT    DOOR    OPEN L/S
      OUT     Y7C  ; MOLD CARINT     PBX045  ON
578   LD      X28  ; RIGHT   DOOR    OPEN L/S
      OR      X7  ; LAMP    TEST
      OUT     Y68  ; RIGHT   DOOR    OPEN    LAMP
581   LD      X33  ; ORIGIN  POSITIONFrom:   ROBOT
      OR      X7  ; LAMP    TEST
      OUT     Y69  ; ROBOT   ORIGIN  LAMP
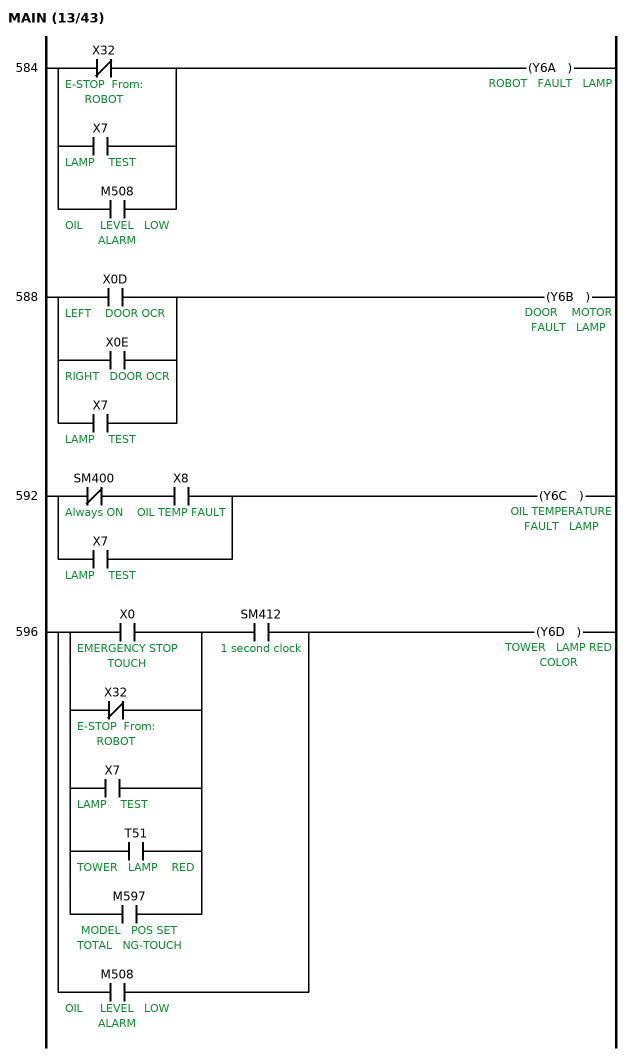
584   LDI     X32  ; E-STOP  From:   ROBOT
      OR      X7  ; LAMP    TEST
      OR      M508  ; OIL     LEVEL   LOW     ALARM
      OUT     Y6A  ; ROBOT   FAULT   LAMP
588   LD      X0D  ; LEFT    DOOR OCR
      OR      X0E  ; RIGHT   DOOR OCR
      OR      X7  ; LAMP    TEST
      OUT     Y6B  ; DOOR    MOTOR   FAULT   LAMP
592   LDI     SM400  ; Always ON
      AND     X8  ; OIL TEMP FAULT
      OR      X7  ; LAMP    TEST
      OUT     Y6C  ; OIL TEMPERATURE FAULT   LAMP
596   LD      X0  ; EMERGENCY STOP  TOUCH
      ORI     X32  ; E-STOP  From:   ROBOT
      OR      X7  ; LAMP    TEST
      OR      T51  ; TOWER   LAMP    RED
      OR      M597  ; MODEL   POS SET TOTAL   NG-TOUCH
      AND     SM412  ; 1 second clock
      OR      M508  ; OIL     LEVEL   LOW     ALARM
      OUT     Y6D  ; TOWER   LAMP RED COLOR
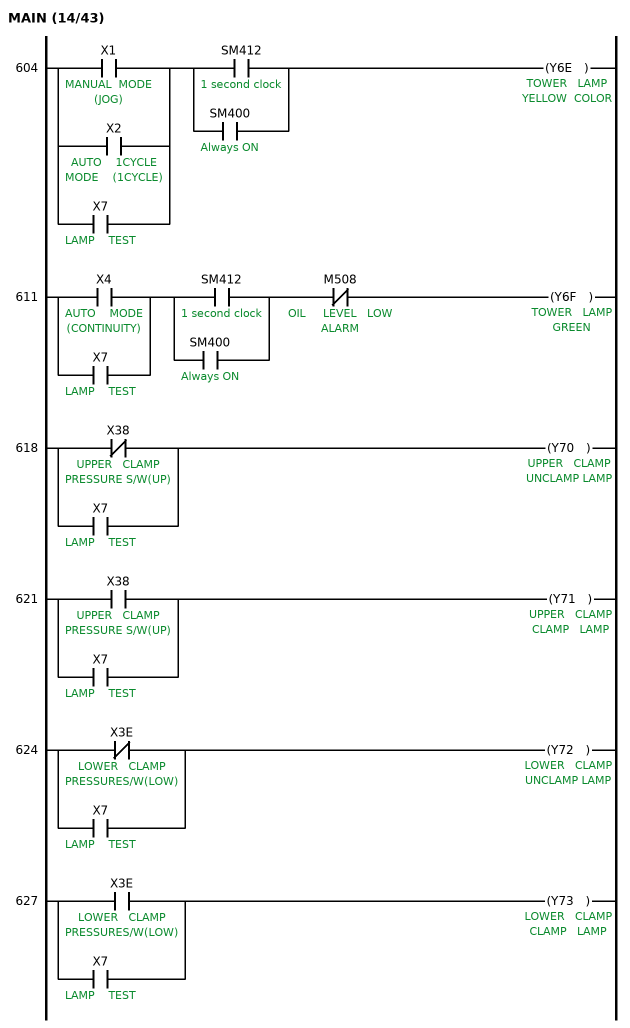
604   LD      X1  ; MANUAL  MODE    (JOG)
      OR      X2  ; AUTO    1CYCLE  MODE    (1CYCLE)
      OR      X7  ; LAMP    TEST
      LD      SM412  ; 1 second clock
      OR      SM400  ; Always ON
      ANB
      OUT     Y6E  ; TOWER   LAMP    YELLOW  COLOR
611   LD      X4  ; AUTO    MODE    (CONTINUITY)
      OR      X7  ; LAMP    TEST
      LD      SM412  ; 1 second clock
      OR      SM400  ; Always ON
      ANB
      ANI     M508  ; OIL     LEVEL   LOW     ALARM
      OUT     Y6F  ; TOWER   LAMP    GREEN
618   LDI     X38  ; UPPER   CLAMP   PRESSURE S/W(UP)
      OR      X7  ; LAMP    TEST
      OUT     Y70  ; UPPER   CLAMP   UNCLAMP LAMP
621   LD      X38  ; UPPER   CLAMP   PRESSURE S/W(UP)
      OR      X7  ; LAMP    TEST
      OUT     Y71  ; UPPER   CLAMP   CLAMP   LAMP
624   LDI     X3E  ; LOWER   CLAMP   PRESSURES/W(LOW)
      OR      X7  ; LAMP    TEST
      OUT     Y72  ; LOWER   CLAMP   UNCLAMP LAMP
627   LD      X3E  ; LOWER   CLAMP   PRESSURES/W(LOW)
      OR      X7  ; LAMP    TEST
      OUT     Y73  ; LOWER   CLAMP   CLAMP   LAMP
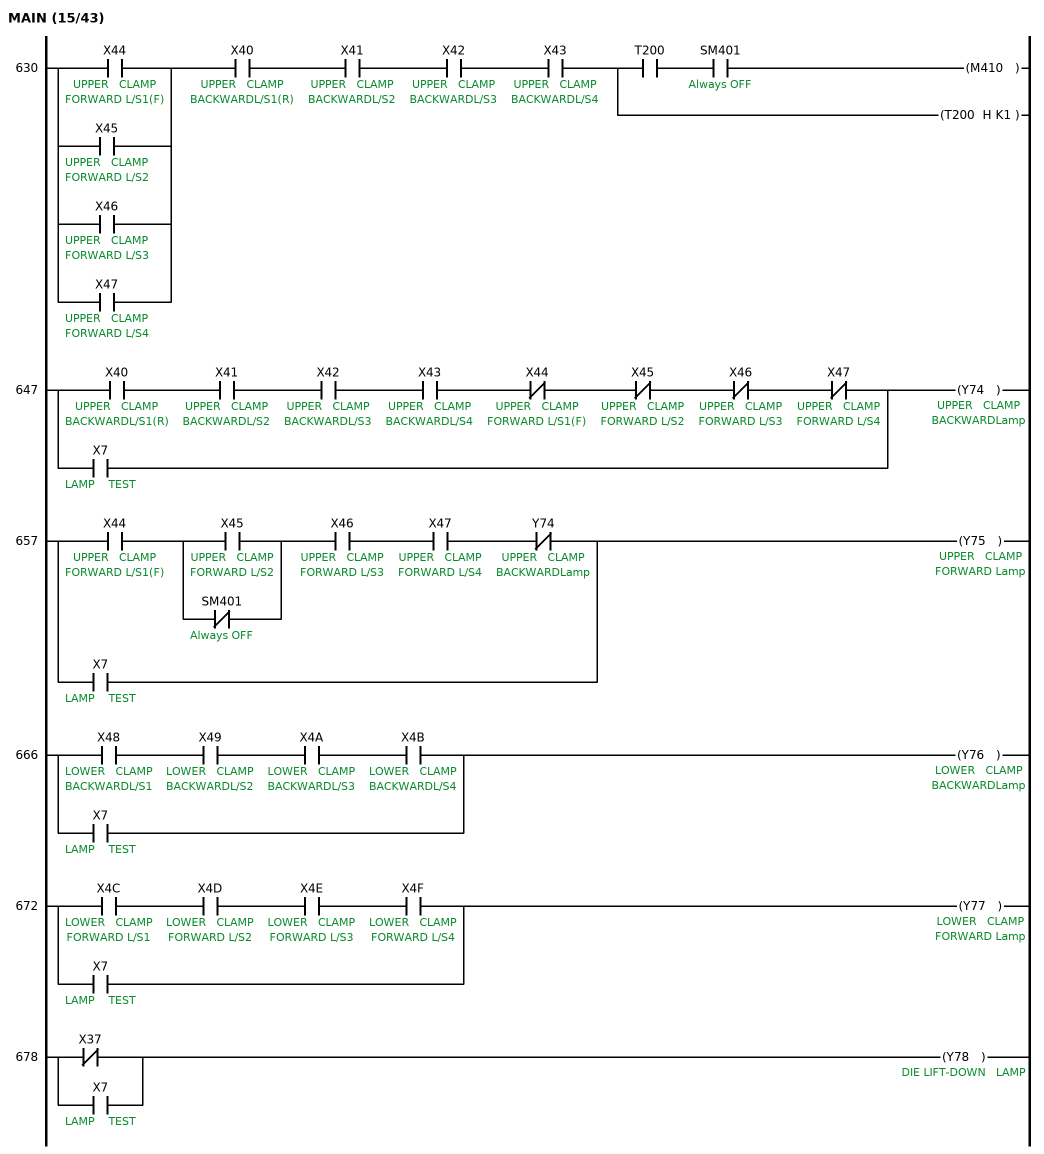
630   LD      X44  ; UPPER   CLAMP   FORWARD L/S1(F)
      OR      X45  ; UPPER   CLAMP   FORWARD L/S2
      OR      X46  ; UPPER   CLAMP   FORWARD L/S3
      OR      X47  ; UPPER   CLAMP   FORWARD L/S4
      AND     X40  ; UPPER   CLAMP   BACKWARDL/S1(R)
      AND     X41  ; UPPER   CLAMP   BACKWARDL/S2
      AND     X42  ; UPPER   CLAMP   BACKWARDL/S3
      AND     X43  ; UPPER   CLAMP   BACKWARDL/S4
      MPS
      AND     T200
      AND     SM401  ; Always OFF
      OUT     M410
      MPP
      OUTH    T200 K1
647   LD      X40  ; UPPER   CLAMP   BACKWARDL/S1(R)
      AND     X41  ; UPPER   CLAMP   BACKWARDL/S2
      AND     X42  ; UPPER   CLAMP   BACKWARDL/S3
      AND     X43  ; UPPER   CLAMP   BACKWARDL/S4
      ANI     X44  ; UPPER   CLAMP   FORWARD L/S1(F)
      ANI     X45  ; UPPER   CLAMP   FORWARD L/S2
      ANI     X46  ; UPPER   CLAMP   FORWARD L/S3
      ANI     X47  ; UPPER   CLAMP   FORWARD L/S4
      OR      X7  ; LAMP    TEST
      OUT     Y74  ; UPPER   CLAMP   BACKWARDLamp
657   LD      X44  ; UPPER   CLAMP   FORWARD L/S1(F)
      LD      X45  ; UPPER   CLAMP   FORWARD L/S2
      ORI     SM401  ; Always OFF
      ANB
      AND     X46  ; UPPER   CLAMP   FORWARD L/S3
      AND     X47  ; UPPER   CLAMP   FORWARD L/S4
      ANI     Y74  ; UPPER   CLAMP   BACKWARDLamp
      OR      X7  ; LAMP    TEST
      OUT     Y75  ; UPPER   CLAMP   FORWARD Lamp
666   LD      X48  ; LOWER   CLAMP   BACKWARDL/S1
      AND     X49  ; LOWER   CLAMP   BACKWARDL/S2
      AND     X4A  ; LOWER   CLAMP   BACKWARDL/S3
      AND     X4B  ; LOWER   CLAMP   BACKWARDL/S4
      OR      X7  ; LAMP    TEST
      OUT     Y76  ; LOWER   CLAMP   BACKWARDLamp
672   LD      X4C  ; LOWER   CLAMP   FORWARD L/S1
      AND     X4D  ; LOWER   CLAMP   FORWARD L/S2
      AND     X4E  ; LOWER   CLAMP   FORWARD L/S3
      AND     X4F  ; LOWER   CLAMP   FORWARD L/S4
      OR      X7  ; LAMP    TEST
      OUT     Y77  ; LOWER   CLAMP   FORWARD Lamp
678   LDI     X37
      OR      X7  ; LAMP    TEST
      OUT     Y78  ; DIE LIFT-DOWN   LAMP
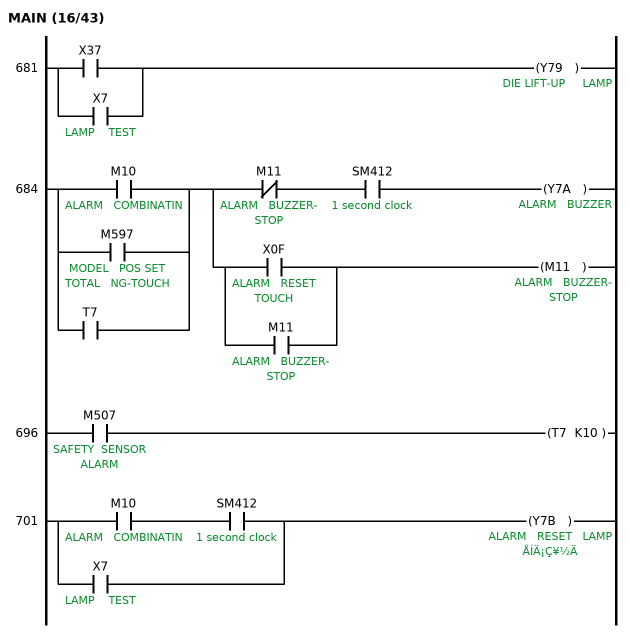
681   LD      X37
      OR      X7  ; LAMP    TEST
      OUT     Y79  ; DIE LIFT-UP     LAMP
684   LD      M10  ; ALARM   COMBINATIN
      OR      M597  ; MODEL   POS SET TOTAL   NG-TOUCH
      OR      T7
      MPS
      ANI     M11  ; ALARM   BUZZER- STOP
      AND     SM412  ; 1 second clock
      OUT     Y7A  ; ALARM   BUZZER
      MPP
      LD      X0F  ; ALARM   RESET   TOUCH
      OR      M11  ; ALARM   BUZZER- STOP
      ANB
      OUT     M11  ; ALARM   BUZZER- STOP
696   LD      M507  ; SAFETY  SENSOR  ALARM
      OUT     T7 K10
701   LD      M10  ; ALARM   COMBINATIN
      AND     SM412  ; 1 second clock
      OR      X7  ; LAMP    TEST
      OUT     Y7B  ; ALARM   RESET   LAMP    ÅÍÄ¡Ç¥½Ã
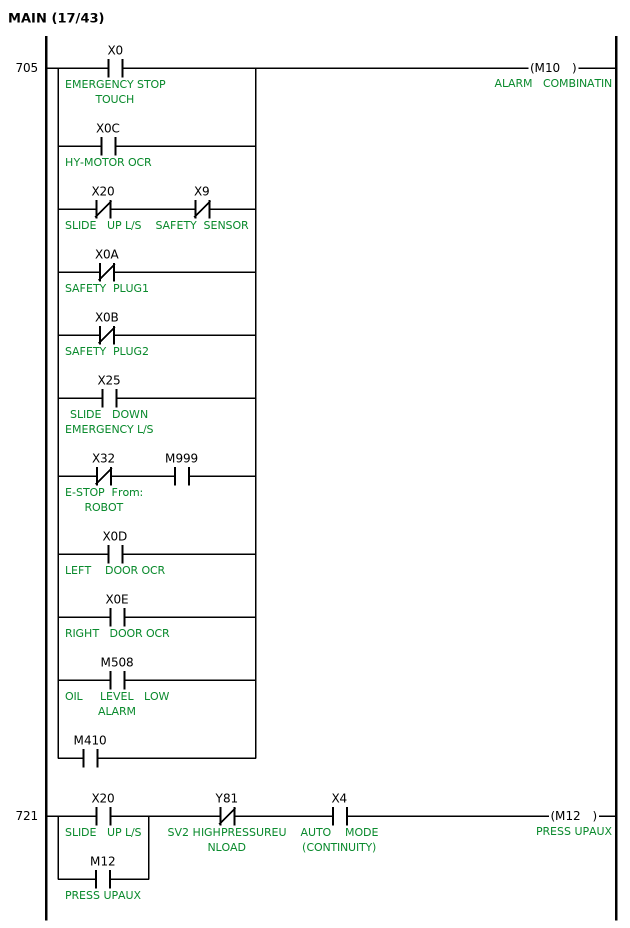
705   LD      X0  ; EMERGENCY STOP  TOUCH
      OR      X0C  ; HY-MOTOR OCR
      LDI     X20  ; SLIDE   UP L/S
      ANI     X9  ; SAFETY  SENSOR
      ORB
      ORI     X0A  ; SAFETY  PLUG1
      ORI     X0B  ; SAFETY  PLUG2
      OR      X25  ; SLIDE   DOWN    EMERGENCY L/S
      LDI     X32  ; E-STOP  From:   ROBOT
      AND     M999
      ORB
      OR      X0D  ; LEFT    DOOR OCR
      OR      X0E  ; RIGHT   DOOR OCR
      OR      M508  ; OIL     LEVEL   LOW     ALARM
      OR      M410
      OUT     M10  ; ALARM   COMBINATIN
721   LD      X20  ; SLIDE   UP L/S
      OR      M12  ; PRESS UPAUX
      ANI     Y81  ; SV2 HIGHPRESSUREUNLOAD
      AND     X4  ; AUTO    MODE    (CONTINUITY)
      OUT     M12  ; PRESS UPAUX
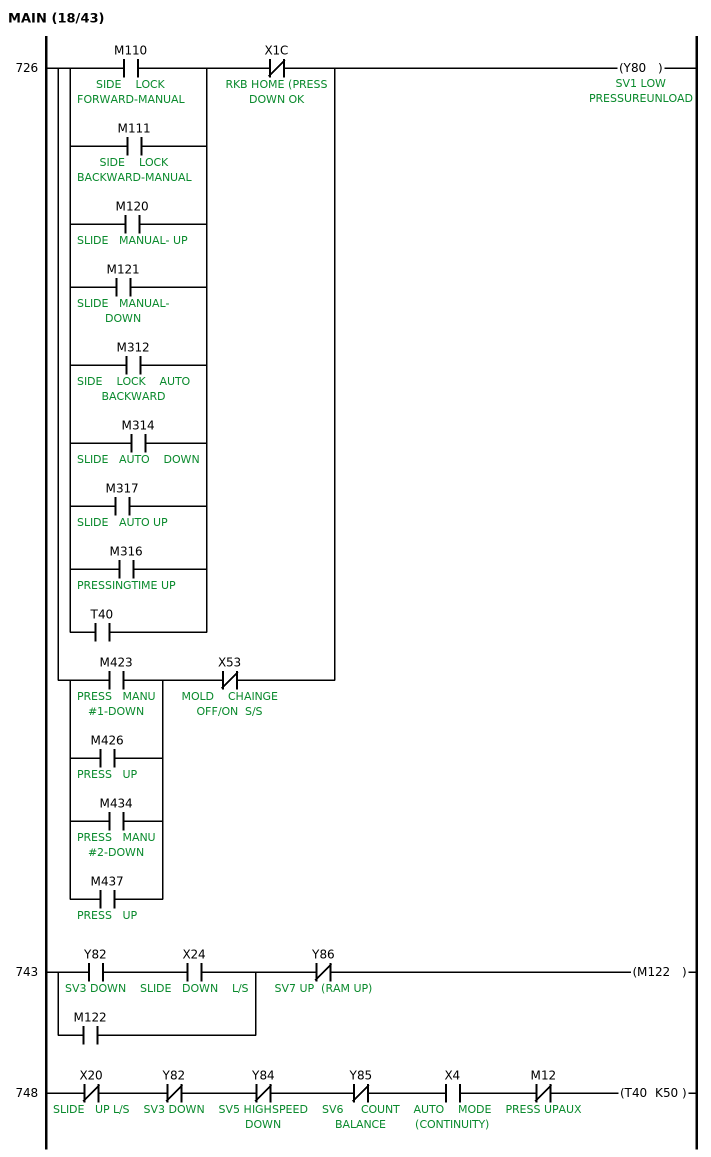
726   LD      M110  ; SIDE    LOCK    FORWARD-MANUAL
      OR      M111  ; SIDE    LOCK    BACKWARD-MANUAL
      OR      M120  ; SLIDE   MANUAL- UP
      OR      M121  ; SLIDE   MANUAL- DOWN
      OR      M312  ; SIDE    LOCK    AUTO    BACKWARD
      OR      M314  ; SLIDE   AUTO    DOWN
      OR      M317  ; SLIDE   AUTO UP
      OR      M316  ; PRESSINGTIME UP
      OR      T40
      ANI     X1C  ; RKB HOME (PRESS DOWN OK
      LD      M423  ; PRESS   MANU #1-DOWN
      OR      M426  ; PRESS   UP
      OR      M434  ; PRESS   MANU #2-DOWN
      OR      M437  ; PRESS   UP
      ANI     X53  ; MOLD    CHAINGE OFF/ON  S/S
      ORB
      OUT     Y80  ; SV1 LOW PRESSUREUNLOAD
743   LD      Y82  ; SV3 DOWN
      AND     X24  ; SLIDE   DOWN    L/S
      OR      M122
      ANI     Y86  ; SV7 UP  (RAM UP)
      OUT     M122
748   LDI     X20  ; SLIDE   UP L/S
      ANI     Y82  ; SV3 DOWN
      ANI     Y84  ; SV5 HIGHSPEED   DOWN
      ANI     Y85  ; SV6     COUNT   BALANCE
      AND     X4  ; AUTO    MODE    (CONTINUITY)
      ANI     M12  ; PRESS UPAUX
      OUT     T40 K50
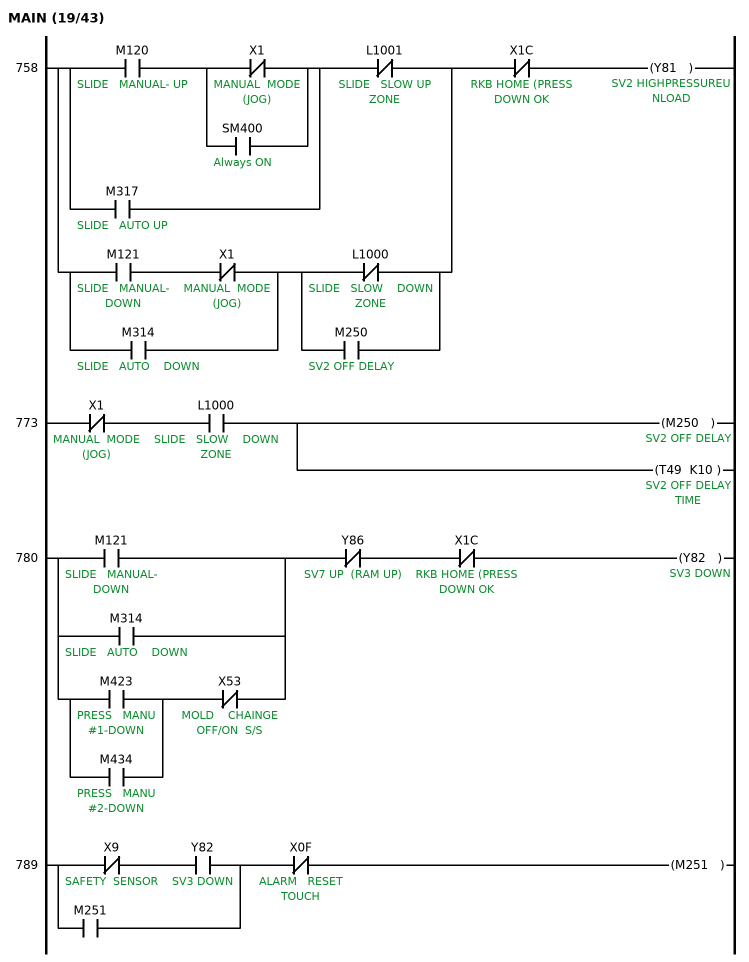
758   LD      M120  ; SLIDE   MANUAL- UP
      LDI     X1  ; MANUAL  MODE    (JOG)
      OR      SM400  ; Always ON
      ANB
      OR      M317  ; SLIDE   AUTO UP
      ANI     L1001  ; SLIDE   SLOW UP ZONE
      LD      M121  ; SLIDE   MANUAL- DOWN
      ANI     X1  ; MANUAL  MODE    (JOG)
      OR      M314  ; SLIDE   AUTO    DOWN
      LDI     L1000  ; SLIDE   SLOW    DOWN    ZONE
      OR      M250  ; SV2 OFF DELAY
      ANB
      ORB
      ANI     X1C  ; RKB HOME (PRESS DOWN OK
      OUT     Y81  ; SV2 HIGHPRESSUREUNLOAD
773   LDI     X1  ; MANUAL  MODE    (JOG)
      AND     L1000  ; SLIDE   SLOW    DOWN    ZONE
      OUT     M250  ; SV2 OFF DELAY
      OUT     T49 K10  ; SV2 OFF DELAY   TIME
780   LD      M121  ; SLIDE   MANUAL- DOWN
      OR      M314  ; SLIDE   AUTO    DOWN
      LD      M423  ; PRESS   MANU #1-DOWN
      OR      M434  ; PRESS   MANU #2-DOWN
      ANI     X53  ; MOLD    CHAINGE OFF/ON  S/S
      ORB
      ANI     Y86  ; SV7 UP  (RAM UP)
      ANI     X1C  ; RKB HOME (PRESS DOWN OK
      OUT     Y82  ; SV3 DOWN
789   LDI     X9  ; SAFETY  SENSOR
      AND     Y82  ; SV3 DOWN
      OR      M251
      ANI     X0F  ; ALARM   RESET   TOUCH
      OUT     M251
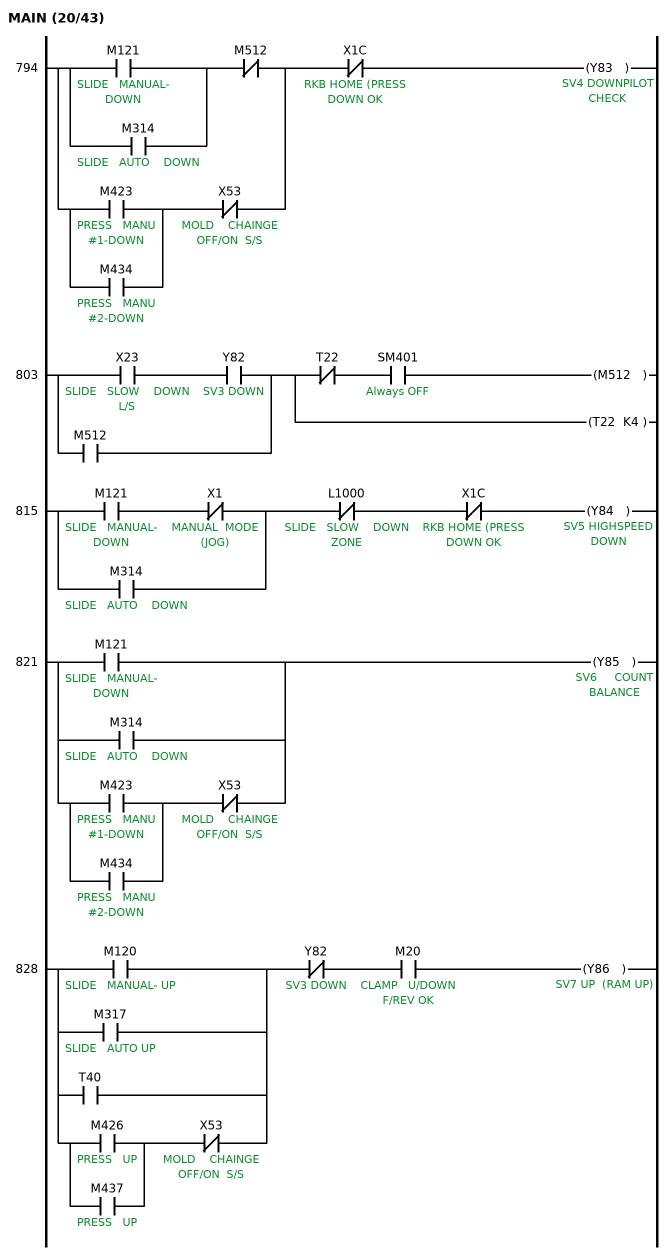
794   LD      M121  ; SLIDE   MANUAL- DOWN
      OR      M314  ; SLIDE   AUTO    DOWN
      ANI     M512
      LD      M423  ; PRESS   MANU #1-DOWN
      OR      M434  ; PRESS   MANU #2-DOWN
      ANI     X53  ; MOLD    CHAINGE OFF/ON  S/S
      ORB
      ANI     X1C  ; RKB HOME (PRESS DOWN OK
      OUT     Y83  ; SV4 DOWNPILOT   CHECK
803   LD      X23  ; SLIDE   SLOW    DOWN L/S
      AND     Y82  ; SV3 DOWN
      OR      M512
      MPS
      ANI     T22
      AND     SM401  ; Always OFF
      OUT     M512
      MPP
      OUT     T22 K4
815   LD      M121  ; SLIDE   MANUAL- DOWN
      ANI     X1  ; MANUAL  MODE    (JOG)
      OR      M314  ; SLIDE   AUTO    DOWN
      ANI     L1000  ; SLIDE   SLOW    DOWN    ZONE
      ANI     X1C  ; RKB HOME (PRESS DOWN OK
      OUT     Y84  ; SV5 HIGHSPEED   DOWN
821   LD      M121  ; SLIDE   MANUAL- DOWN
      OR      M314  ; SLIDE   AUTO    DOWN
      LD      M423  ; PRESS   MANU #1-DOWN
      OR      M434  ; PRESS   MANU #2-DOWN
      ANI     X53  ; MOLD    CHAINGE OFF/ON  S/S
      ORB
      OUT     Y85  ; SV6     COUNT   BALANCE
828   LD      M120  ; SLIDE   MANUAL- UP
      OR      M317  ; SLIDE   AUTO UP
      OR      T40
      LD      M426  ; PRESS   UP
      OR      M437  ; PRESS   UP
      ANI     X53  ; MOLD    CHAINGE OFF/ON  S/S
      ORB
      ANI     Y82  ; SV3 DOWN
      AND     M20  ; CLAMP   U/DOWN  F/REV OK
      OUT     Y86  ; SV7 UP  (RAM UP)
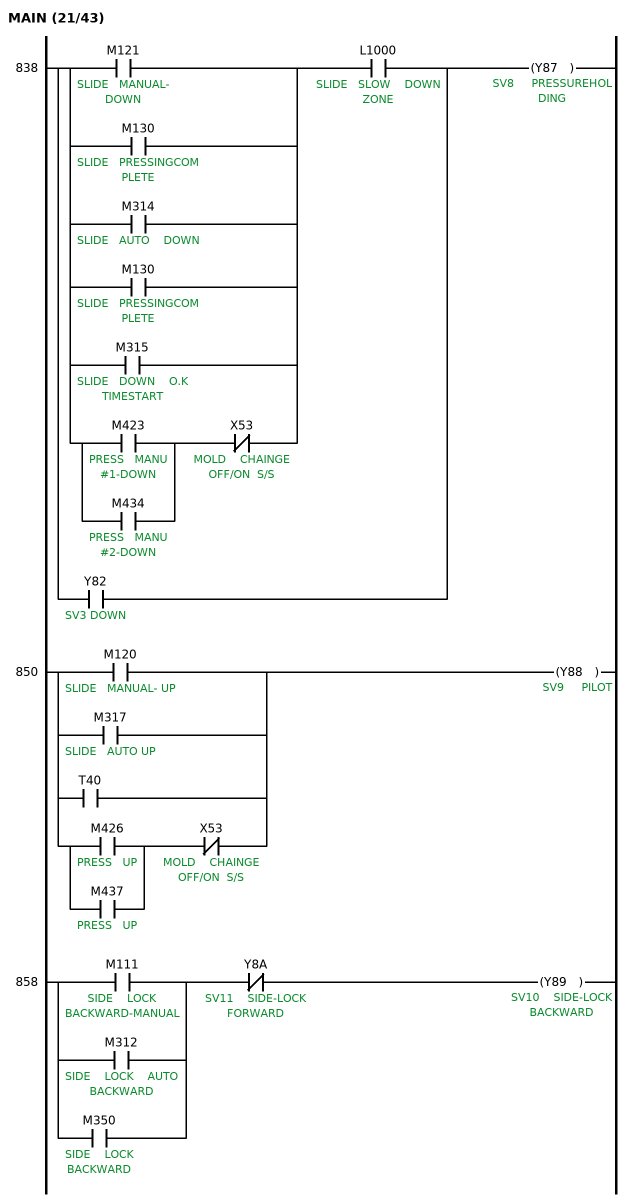
838   LD      M121  ; SLIDE   MANUAL- DOWN
      OR      M130  ; SLIDE   PRESSINGCOMPLETE
      OR      M314  ; SLIDE   AUTO    DOWN
      OR      M130  ; SLIDE   PRESSINGCOMPLETE
      OR      M315  ; SLIDE   DOWN    O.K TIMESTART
      LD      M423  ; PRESS   MANU #1-DOWN
      OR      M434  ; PRESS   MANU #2-DOWN
      ANI     X53  ; MOLD    CHAINGE OFF/ON  S/S
      ORB
      AND     L1000  ; SLIDE   SLOW    DOWN    ZONE
      OR      Y82  ; SV3 DOWN
      OUT     Y87  ; SV8     PRESSUREHOLDING
850   LD      M120  ; SLIDE   MANUAL- UP
      OR      M317  ; SLIDE   AUTO UP
      OR      T40
      LD      M426  ; PRESS   UP
      OR      M437  ; PRESS   UP
      ANI     X53  ; MOLD    CHAINGE OFF/ON  S/S
      ORB
      OUT     Y88  ; SV9     PILOT
858   LD      M111  ; SIDE    LOCK    BACKWARD-MANUAL
      OR      M312  ; SIDE    LOCK    AUTO    BACKWARD
      OR      M350  ; SIDE    LOCK    BACKWARD
      ANI     Y8A  ; SV11    SIDE-LOCK       FORWARD
      OUT     Y89  ; SV10    SIDE-LOCK       BACKWARD
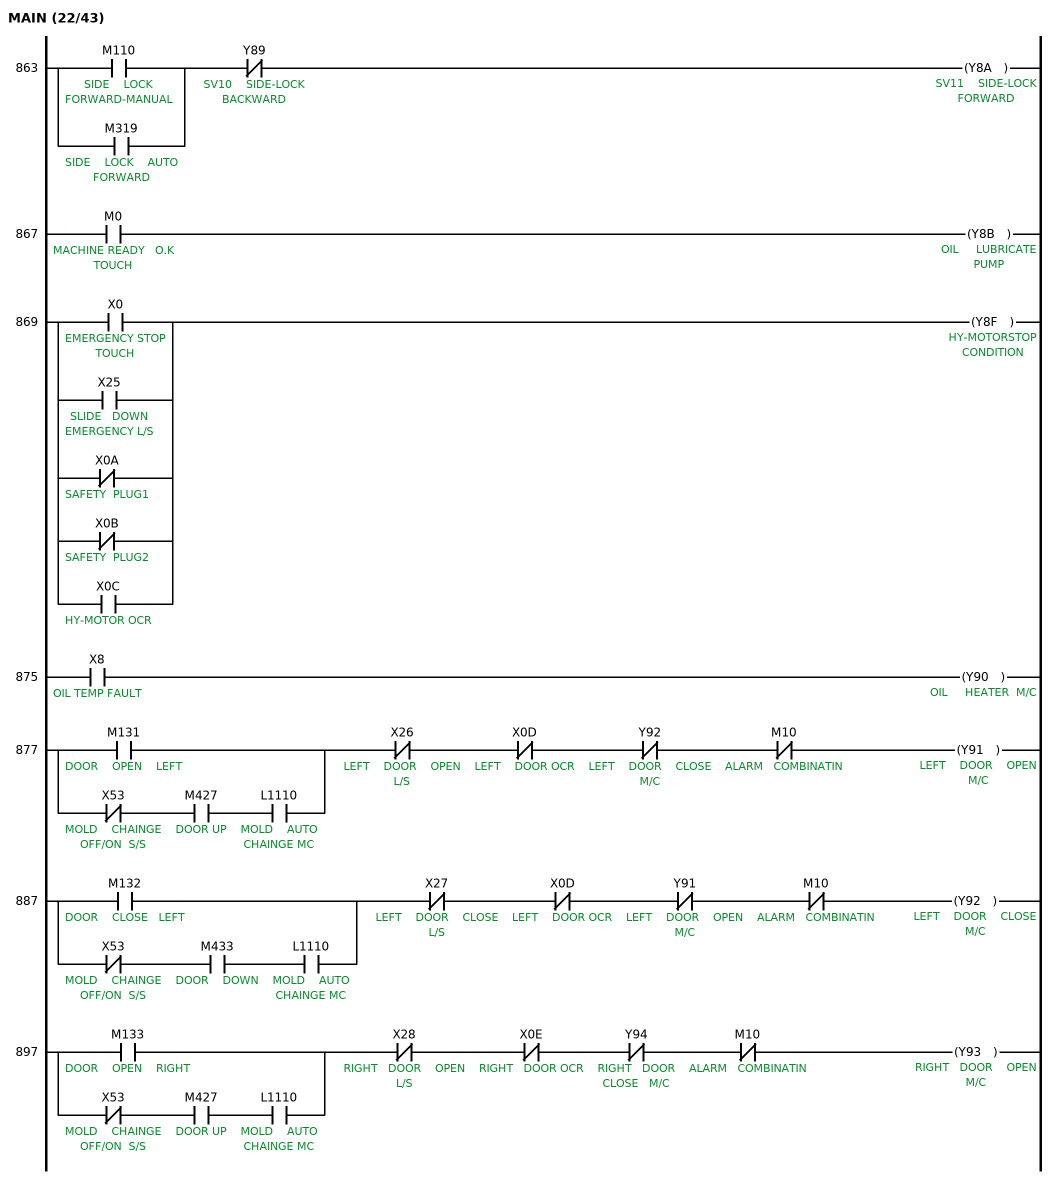
863   LD      M110  ; SIDE    LOCK    FORWARD-MANUAL
      OR      M319  ; SIDE    LOCK    AUTO    FORWARD
      ANI     Y89  ; SV10    SIDE-LOCK       BACKWARD
      OUT     Y8A  ; SV11    SIDE-LOCK       FORWARD
867   LD      M0  ; MACHINE READY   O.K     TOUCH
      OUT     Y8B  ; OIL     LUBRICATE       PUMP
869   LD      X0  ; EMERGENCY STOP  TOUCH
      OR      X25  ; SLIDE   DOWN    EMERGENCY L/S
      ORI     X0A  ; SAFETY  PLUG1
      ORI     X0B  ; SAFETY  PLUG2
      OR      X0C  ; HY-MOTOR OCR
      OUT     Y8F  ; HY-MOTORSTOP    CONDITION
875   LD      X8  ; OIL TEMP FAULT
      OUT     Y90  ; OIL     HEATER  M/C
877   LD      M131  ; DOOR    OPEN    LEFT
      LDI     X53  ; MOLD    CHAINGE OFF/ON  S/S
      AND     M427  ; DOOR UP
      AND     L1110  ; MOLD    AUTO    CHAINGE MC
      ORB
      ANI     X26  ; LEFT    DOOR    OPEN L/S
      ANI     X0D  ; LEFT    DOOR OCR
      ANI     Y92  ; LEFT    DOOR    CLOSE   M/C
      ANI     M10  ; ALARM   COMBINATIN
      OUT     Y91  ; LEFT    DOOR    OPEN M/C
887   LD      M132  ; DOOR    CLOSE   LEFT
      LDI     X53  ; MOLD    CHAINGE OFF/ON  S/S
      AND     M433  ; DOOR    DOWN
      AND     L1110  ; MOLD    AUTO    CHAINGE MC
      ORB
      ANI     X27  ; LEFT    DOOR    CLOSE   L/S
      ANI     X0D  ; LEFT    DOOR OCR
      ANI     Y91  ; LEFT    DOOR    OPEN M/C
      ANI     M10  ; ALARM   COMBINATIN
      OUT     Y92  ; LEFT    DOOR    CLOSE   M/C
897   LD      M133  ; DOOR    OPEN    RIGHT
      LDI     X53  ; MOLD    CHAINGE OFF/ON  S/S
      AND     M427  ; DOOR UP
      AND     L1110  ; MOLD    AUTO    CHAINGE MC
      ORB
      ANI     X28  ; RIGHT   DOOR    OPEN L/S
      ANI     X0E  ; RIGHT   DOOR OCR
      ANI     Y94  ; RIGHT   DOOR    CLOSE   M/C
      ANI     M10  ; ALARM   COMBINATIN
      OUT     Y93  ; RIGHT   DOOR    OPEN    M/C
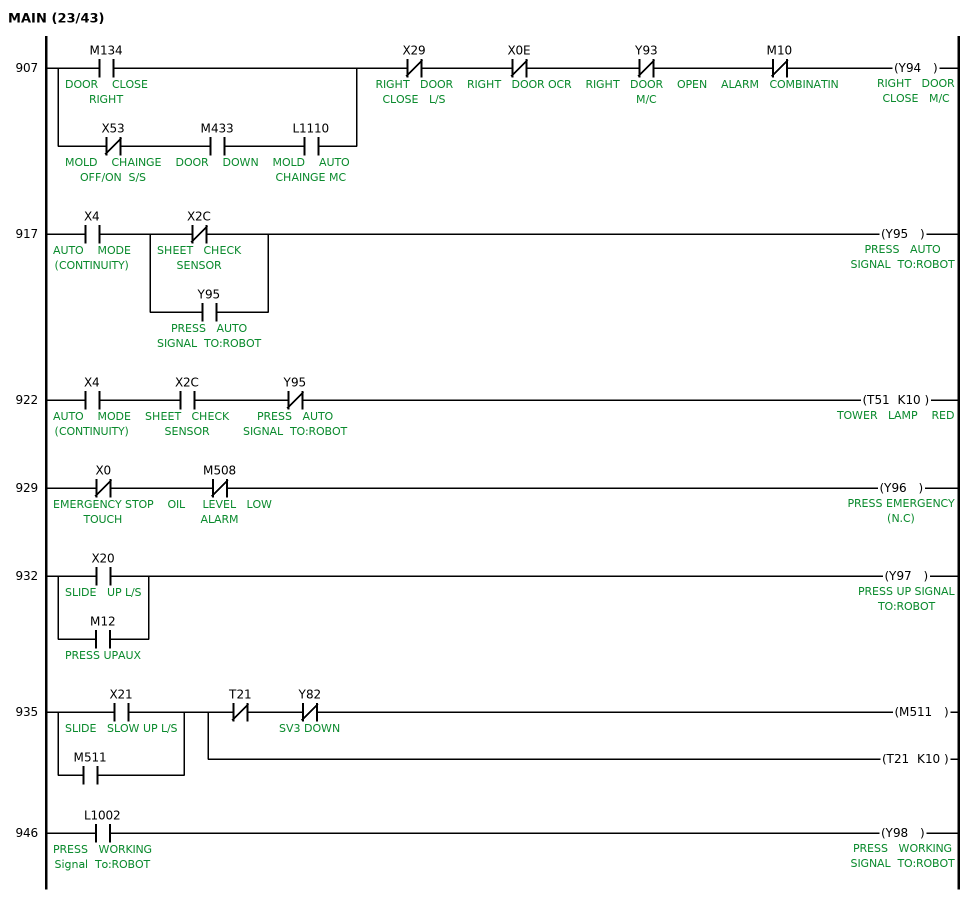
907   LD      M134  ; DOOR    CLOSE   RIGHT
      LDI     X53  ; MOLD    CHAINGE OFF/ON  S/S
      AND     M433  ; DOOR    DOWN
      AND     L1110  ; MOLD    AUTO    CHAINGE MC
      ORB
      ANI     X29  ; RIGHT   DOOR    CLOSE   L/S
      ANI     X0E  ; RIGHT   DOOR OCR
      ANI     Y93  ; RIGHT   DOOR    OPEN    M/C
      ANI     M10  ; ALARM   COMBINATIN
      OUT     Y94  ; RIGHT   DOOR    CLOSE   M/C
917   LD      X4  ; AUTO    MODE    (CONTINUITY)
      LDI     X2C  ; SHEET   CHECK   SENSOR
      OR      Y95  ; PRESS   AUTO    SIGNAL  TO:ROBOT
      ANB
      OUT     Y95  ; PRESS   AUTO    SIGNAL  TO:ROBOT
922   LD      X4  ; AUTO    MODE    (CONTINUITY)
      AND     X2C  ; SHEET   CHECK   SENSOR
      ANI     Y95  ; PRESS   AUTO    SIGNAL  TO:ROBOT
      OUT     T51 K10  ; TOWER   LAMP    RED
929   LDI     X0  ; EMERGENCY STOP  TOUCH
      ANI     M508  ; OIL     LEVEL   LOW     ALARM
      OUT     Y96  ; PRESS EMERGENCY (N.C)
932   LD      X20  ; SLIDE   UP L/S
      OR      M12  ; PRESS UPAUX
      OUT     Y97  ; PRESS UP SIGNAL TO:ROBOT
935   LD      X21  ; SLIDE   SLOW UP L/S
      OR      M511
      MPS
      ANI     T21
      ANI     Y82  ; SV3 DOWN
      OUT     M511
      MPP
      OUT     T21 K10
946   LD      L1002  ; PRESS   WORKING Signal  To:ROBOT
      OUT     Y98  ; PRESS   WORKING SIGNAL  TO:ROBOT
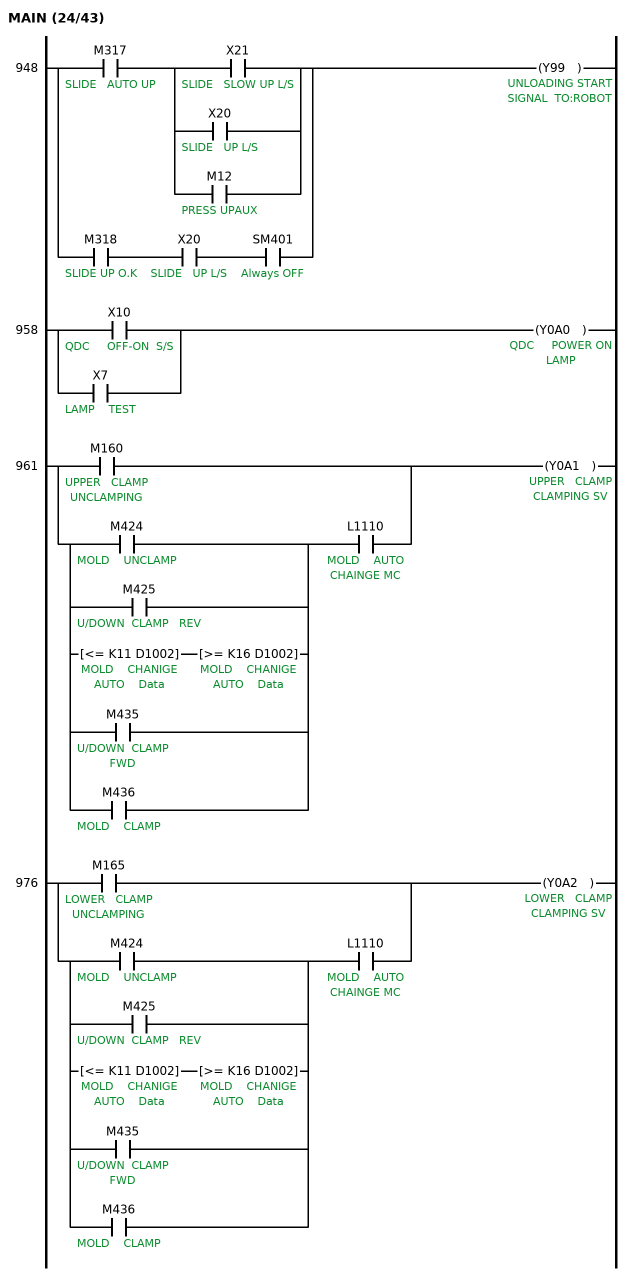
948   LD      M317  ; SLIDE   AUTO UP
      LD      X21  ; SLIDE   SLOW UP L/S
      OR      X20  ; SLIDE   UP L/S
      OR      M12  ; PRESS UPAUX
      ANB
      LD      M318  ; SLIDE UP O.K
      AND     X20  ; SLIDE   UP L/S
      AND     SM401  ; Always OFF
      ORB
      OUT     Y99  ; UNLOADING START SIGNAL  TO:ROBOT
958   LD      X10  ; QDC     OFF-ON  S/S
      OR      X7  ; LAMP    TEST
      OUT     Y0A0  ; QDC     POWER ON LAMP
961   LD      M160  ; UPPER   CLAMP   UNCLAMPING
      LD      M424  ; MOLD    UNCLAMP
      OR      M425  ; U/DOWN  CLAMP   REV
      LD<=    K11 D1002  ; MOLD    CHANIGE AUTO    Data
      AND>=   K16 D1002  ; MOLD    CHANIGE AUTO    Data
      ORB
      OR      M435  ; U/DOWN  CLAMP   FWD
      OR      M436  ; MOLD    CLAMP
      AND     L1110  ; MOLD    AUTO    CHAINGE MC
      ORB
      OUT     Y0A1  ; UPPER   CLAMP   CLAMPING SV
976   LD      M165  ; LOWER   CLAMP   UNCLAMPING
      LD      M424  ; MOLD    UNCLAMP
      OR      M425  ; U/DOWN  CLAMP   REV
      LD<=    K11 D1002  ; MOLD    CHANIGE AUTO    Data
      AND>=   K16 D1002  ; MOLD    CHANIGE AUTO    Data
      ORB
      OR      M435  ; U/DOWN  CLAMP   FWD
      OR      M436  ; MOLD    CLAMP
      AND     L1110  ; MOLD    AUTO    CHAINGE MC
      ORB
      OUT     Y0A2  ; LOWER   CLAMP   CLAMPING SV
